   CamCalc.CrossChain_Cam[0..99].inflectionPointParameter := 0.5;
   CamCalc.CrossChain_Cam[0..99].modVeloTrapezoidParameter := 1.0;
   CamCalc.CrossChain_Cam[0..99].modSineMaxAccelCaStar := 0.0;
   CamCalc.CrossChain_Cam[0].camProfileType := 2;
   CamCalc.CrossChain_Cam[1..2].camProfileType := 1;
   CamCalc.CrossChain_Cam[3].camProfileType := 3;
   CamCalc.CrossChain_Cam[4..5].camProfileType := 1;
   CamCalc.CrossChain_Cam[6..99].camProfileType := 0;
   CamCalc.BeltChain_Cam[0..99].leadingValueStart := 0.0;
   CamCalc.BeltChain_Cam[0..99].leadingValueEnd := 0.0;
   CamCalc.BeltChain_Cam[0..99].followingValueStart := 0.0;
   CamCalc.BeltChain_Cam[0..99].followingValueEnd := 0.0;
   CamCalc.BeltChain_Cam[0..99].geoVeloStart := 0.0;
   CamCalc.BeltChain_Cam[0..99].geoVeloEnd := 0.0;
   CamCalc.BeltChain_Cam[0..99].geoAccelStart := 0.0;
   CamCalc.BeltChain_Cam[0..99].geoAccelEnd := 0.0;
   CamCalc.BeltChain_Cam[0..99].geoJerkStart := 0.0;
   CamCalc.BeltChain_Cam[0..99].geoJerkEnd := 0.0;
   CamCalc.BeltChain_Cam[0..99].inflectionPointParameter := 0.5;
   CamCalc.BeltChain_Cam[0..99].modVeloTrapezoidParameter := 1.0;
   CamCalc.BeltChain_Cam[0..99].modSineMaxAccelCaStar := 0.0;
   CamCalc.BeltChain_Cam[0..99].camProfileType := 0;
   CamCalc.ContChain_Cam[0..99].leadingValueStart := 0.0;
   CamCalc.ContChain_Cam[0].leadingValueEnd := 360.0;
   CamCalc.ContChain_Cam[1..99].leadingValueEnd := 0.0;
   CamCalc.ContChain_Cam[0..99].followingValueStart := 0.0;
   CamCalc.ContChain_Cam[0].followingValueEnd := 406.399993896484;
   CamCalc.ContChain_Cam[1..99].followingValueEnd := 0.0;
   CamCalc.ContChain_Cam[0..99].geoVeloStart := 0.0;
   CamCalc.ContChain_Cam[0..99].geoVeloEnd := 0.0;
   CamCalc.ContChain_Cam[0..99].geoAccelStart := 0.0;
   CamCalc.ContChain_Cam[0..99].geoAccelEnd := 0.0;
   CamCalc.ContChain_Cam[0..99].geoJerkStart := 0.0;
   CamCalc.ContChain_Cam[0..99].geoJerkEnd := 0.0;
   CamCalc.ContChain_Cam[0..99].inflectionPointParameter := 0.5;
   CamCalc.ContChain_Cam[0..99].modVeloTrapezoidParameter := 1.0;
   CamCalc.ContChain_Cam[0..99].modSineMaxAccelCaStar := 0.0;
   CamCalc.ContChain_Cam[0].camProfileType := 3;
   CamCalc.ContChain_Cam[1..99].camProfileType := 0;
   CamCalc.TransferChain_Cam[0..99].leadingValueStart := 0.0;
   CamCalc.TransferChain_Cam[0..99].leadingValueEnd := 0.0;
   CamCalc.TransferChain_Cam[0..99].followingValueStart := 0.0;
   CamCalc.TransferChain_Cam[0..99].followingValueEnd := 0.0;
   CamCalc.TransferChain_Cam[0..99].geoVeloStart := 0.0;
   CamCalc.TransferChain_Cam[0..99].geoVeloEnd := 0.0;
   CamCalc.TransferChain_Cam[0..99].geoAccelStart := 0.0;
   CamCalc.TransferChain_Cam[0..99].geoAccelEnd := 0.0;
   CamCalc.TransferChain_Cam[0..99].geoJerkStart := 0.0;
   CamCalc.TransferChain_Cam[0..99].geoJerkEnd := 0.0;
   CamCalc.TransferChain_Cam[0..99].inflectionPointParameter := 0.5;
   CamCalc.TransferChain_Cam[0..99].modVeloTrapezoidParameter := 1.0;
   CamCalc.TransferChain_Cam[0..99].modSineMaxAccelCaStar := 0.0;
   CamCalc.TransferChain_Cam[0..99].camProfileType := 0;
   CamCalc.ColumnAscChain_Cam[0..99].leadingValueStart := 0.0;
   CamCalc.ColumnAscChain_Cam[0..99].leadingValueEnd := 0.0;
   CamCalc.ColumnAscChain_Cam[0..99].followingValueStart := 0.0;
   CamCalc.ColumnAscChain_Cam[0..99].followingValueEnd := 0.0;
   CamCalc.ColumnAscChain_Cam[0..99].geoVeloStart := 0.0;
   CamCalc.ColumnAscChain_Cam[0..99].geoVeloEnd := 0.0;
   CamCalc.ColumnAscChain_Cam[0..99].geoAccelStart := 0.0;
   CamCalc.ColumnAscChain_Cam[0..99].geoAccelEnd := 0.0;
   CamCalc.ColumnAscChain_Cam[0..99].geoJerkStart := 0.0;
   CamCalc.ColumnAscChain_Cam[0..99].geoJerkEnd := 0.0;
   CamCalc.ColumnAscChain_Cam[0..99].inflectionPointParameter := 0.5;
   CamCalc.ColumnAscChain_Cam[0..99].modVeloTrapezoidParameter := 1.0;
   CamCalc.ColumnAscChain_Cam[0..99].modSineMaxAccelCaStar := 0.0;
   CamCalc.ColumnAscChain_Cam[0..99].camProfileType := 0;
   CamCalc.ColumnDescChain_Cam[0..99].leadingValueStart := 0.0;
   CamCalc.ColumnDescChain_Cam[0..99].leadingValueEnd := 0.0;
   CamCalc.ColumnDescChain_Cam[0..99].followingValueStart := 0.0;
   CamCalc.ColumnDescChain_Cam[0..99].followingValueEnd := 0.0;
   CamCalc.ColumnDescChain_Cam[0..99].geoVeloStart := 0.0;
   CamCalc.ColumnDescChain_Cam[0..99].geoVeloEnd := 0.0;
   CamCalc.ColumnDescChain_Cam[0..99].geoAccelStart := 0.0;
   CamCalc.ColumnDescChain_Cam[0..99].geoAccelEnd := 0.0;
   CamCalc.ColumnDescChain_Cam[0..99].geoJerkStart := 0.0;
   CamCalc.ColumnDescChain_Cam[0..99].geoJerkEnd := 0.0;
   CamCalc.ColumnDescChain_Cam[0..99].inflectionPointParameter := 0.5;
   CamCalc.ColumnDescChain_Cam[0..99].modVeloTrapezoidParameter := 1.0;
   CamCalc.ColumnDescChain_Cam[0..99].modSineMaxAccelCaStar := 0.0;
   CamCalc.ColumnDescChain_Cam[0..99].camProfileType := 0;
   CamCalc.CrossChain4_Cam[0].leadingValueStart := 0.0;
   CamCalc.CrossChain4_Cam[1].leadingValueStart := 193.679992675781;
   CamCalc.CrossChain4_Cam[2..3].leadingValueStart := 225.360000610352;
   CamCalc.CrossChain4_Cam[4].leadingValueStart := 328.320007324219;
   CamCalc.CrossChain4_Cam[5].leadingValueStart := 360.0;
   CamCalc.CrossChain4_Cam[6..99].leadingValueStart := 0.0;
   CamCalc.CrossChain4_Cam[0].leadingValueEnd := 162.0;
   CamCalc.CrossChain4_Cam[1..2].leadingValueEnd := 0.0;
   CamCalc.CrossChain4_Cam[3].leadingValueEnd := 296.640014648438;
   CamCalc.CrossChain4_Cam[4..99].leadingValueEnd := 0.0;
   CamCalc.CrossChain4_Cam[0].followingValueStart := 0.0;
   CamCalc.CrossChain4_Cam[1].followingValueStart := 31.8745098114014;
   CamCalc.CrossChain4_Cam[2..3].followingValueStart := 191.247055053711;
   CamCalc.CrossChain4_Cam[4].followingValueStart := 780.925476074219;
   CamCalc.CrossChain4_Cam[5].followingValueStart := 812.799987792969;
   CamCalc.CrossChain4_Cam[6..99].followingValueStart := 0.0;
   CamCalc.CrossChain4_Cam[0..2].followingValueEnd := 0.0;
   CamCalc.CrossChain4_Cam[3].followingValueEnd := 621.552917480469;
   CamCalc.CrossChain4_Cam[4..99].followingValueEnd := 0.0;
   CamCalc.CrossChain4_Cam[0..99].geoVeloStart := 0.0;
   CamCalc.CrossChain4_Cam[0..99].geoVeloEnd := 0.0;
   CamCalc.CrossChain4_Cam[0..99].geoAccelStart := 0.0;
   CamCalc.CrossChain4_Cam[0..99].geoAccelEnd := 0.0;
   CamCalc.CrossChain4_Cam[0..99].geoJerkStart := 0.0;
   CamCalc.CrossChain4_Cam[0..99].geoJerkEnd := 0.0;
   CamCalc.CrossChain4_Cam[0..99].inflectionPointParameter := 0.5;
   CamCalc.CrossChain4_Cam[0..99].modVeloTrapezoidParameter := 1.0;
   CamCalc.CrossChain4_Cam[0..99].modSineMaxAccelCaStar := 0.0;
   CamCalc.CrossChain4_Cam[0].camProfileType := 2;
   CamCalc.CrossChain4_Cam[1..2].camProfileType := 1;
   CamCalc.CrossChain4_Cam[3].camProfileType := 3;
   CamCalc.CrossChain4_Cam[4..5].camProfileType := 1;
   CamCalc.CrossChain4_Cam[6..99].camProfileType := 0;
   Chain1Long.AlmOk := TRUE;
   Chain1Long.StationWorked := TRUE;
   Chain1Long.CheckObstruction := TRUE;
   Chain1Long.OutChainObstruction := TRUE;
   Chain1Long.StrobeWork := FALSE;
   Chain1Long.StrobeShift := FALSE;
   Chain1Long.ManualMovement := FALSE;
   Chain1Long.OkToStop := TRUE;
   Chain1Long.PosOk := FALSE;
   Chain1Long.Ons_PosOk := FALSE;
   Chain1Long.EnaMove := TRUE;
   Chain1Long.StationEna := FALSE;
   Chain1Long.ModeLong := TRUE;
   Chain1Long.ModeCross := FALSE;
   Chain1Long.ModeCont := FALSE;
   Chain1Long.Cfg_Mould_ChainSteps := 1;
   Chain1Long.Cfg_Mould_EndPos := 38;
   Chain1Long.Shift_Lenght := 39;
   Chain1Long.PosMasterAdvanceStep := 0.0;
   Chain1Long.Input.EndChaMouPre := FALSE;
   Chain1Long.Input.PshHig := FALSE;
   Chain1Long.Input.PshLow := FALSE;
   Chain1Long.Output.PshHig := FALSE;
   Chain1Long.Output.PshLow := FALSE;
   Chain1Long.Man.EnaPbt := FALSE;
   Chain1Long.Man.RstCmd := TRUE;
   Chain1Long.Man.ScreenNumber := 300_010_301;
   Chain1Long.Man.WithinScreenRange := 0;
   Chain1Long.Drive.AlmOk := FALSE;
   Chain1Long.Drive.AlmEmerg := FALSE;
   Chain1Long.Drive.AlmNode := FALSE;
   Chain1Long.Drive.InitPosDrive := FALSE;
   Chain1Long.Drive.InitPosDrivePLS := FALSE;
   Chain1Long.Drive.GearingON := FALSE;
   Chain1Long.Drive.CamHook := FALSE;
   Chain1Long.Drive.CamStoppingPhase := FALSE;
   Chain1Long.Drive.RepositioningRequest := FALSE;
   Chain1Long.Drive.CamRequestResult := FALSE;
   Chain1Long.Drive.CamRequestError := FALSE;
   Chain1Long.Drive.CamRequestOk := TRUE;
   Chain1Long.Drive.CalibDisAxisReq := FALSE;
   Chain1Long.Drive.CalibReq := FALSE;
   Chain1Long.Drive.CalibProcess := FALSE;
   Chain1Long.Drive.HwOvertravelDisReq := FALSE;
   Chain1Long.Drive.HwOvertravelEnReq := FALSE;
   Chain1Long.Drive.AuxCamRequest := FALSE;
   Chain1Long.Drive.TorquePeakEna := TRUE;
   Chain1Long.Drive.Cmd_Repos := FALSE;
   Chain1Long.Drive.Ons_CamRequest := FALSE;
   Chain1Long.Drive.AuxCmdPosition := 0;
   Chain1Long.Drive.Unwind := 406.4;
   Chain1Long.Drive.MaxDev := 150.0;
   Chain1Long.Drive.ReposSpeed := 10.0;
   Chain1Long.Drive.CalcSlaveDifferenceABS := 0.0;
   Chain1Long.Drive.CalcModPosition := 0.0;
   Chain1Long.Drive.CalcSlaveDifference := 0.0;
   Chain1Long.Drive.CalcMinDeltaPos := 0.0;
   Chain1Long.Drive.CalcMaxDeltaPos := 0.0;
   Chain1Long.Drive.CalcHalfPosUnwind := 0.0;
   Chain1Long.Drive.Man.Cmd_PosJog := FALSE;
   Chain1Long.Drive.Man.Cmd_NegJog := FALSE;
   Chain1Long.Drive.Man.Cmd_Step := FALSE;
   Chain1Long.Drive.Man.Cmd_Forward := FALSE;
   Chain1Long.Drive.Man.Cmd_Backward := FALSE;
   Chain1Long.Drive.Man.Cmd_Up := FALSE;
   Chain1Long.Drive.Man.Cmd_Down := FALSE;
   Chain1Long.Drive.Man.Cmd_Intermediate := FALSE;
   Chain1Long.Drive.Man.Cmd_Open := FALSE;
   Chain1Long.Drive.Man.Cmd_Close := FALSE;
   Chain1Long.Drive.Man.Cmd_PreOpen := FALSE;
   Chain1Long.Drive.Man.Cmd_Maintenance := FALSE;
   Chain1Long.Drive.Man.Cmd_OperatorSide := FALSE;
   Chain1Long.Drive.Man.Cmd_NotOperatorSide := FALSE;
   Chain1Long.Drive.Man.Cmd_OnMould := FALSE;
   Chain1Long.Drive.Man.Cmd_OffMould := FALSE;
   Chain1Long.Drive.Man.Cmd_Pos0 := FALSE;
   Chain1Long.Drive.Man.Cmd_Pos1 := FALSE;
   Chain1Long.Drive.Man.Cmd_Pos2 := FALSE;
   Chain1Long.Drive.Man.Cmd_Pos3 := FALSE;
   Chain1Long.Drive.Man.Cmd_Pos4 := FALSE;
   Chain1Long.Drive.Man.Cmd_Pos5 := FALSE;
   Chain1Long.Drive.Man.Ons_Step := FALSE;
   Chain1Long.Drive.Man.PhaseJogCmd := FALSE;
   Chain1Long.Drive.Man.CmdStartStep := FALSE;
   Chain1Long.Drive.Man.CmdEndStep := FALSE;
   Chain1Long.Drive.Man.StepCond := FALSE;
   Chain1Long.Drive.Man.TON_DelayHomeCmd.PT := T#3S;
   Chain1Long.Drive.Man.TON_DelayHomeCmd.IN := FALSE;
   Chain1Long.Drive.Auto.Cmd_Step := FALSE;
   Chain1Long.Drive.Auto.Cmd_StartStep := FALSE;
   Chain1Long.Drive.Auto.Cmd_EndStep := FALSE;
   Chain1Long.Drive.Auto.Cmd_Forward := FALSE;
   Chain1Long.Drive.Auto.Cmd_Backward := FALSE;
   Chain1Long.Drive.Auto.Cmd_Up := FALSE;
   Chain1Long.Drive.Auto.Cmd_Down := FALSE;
   Chain1Long.Drive.Auto.Cmd_Intermediate := FALSE;
   Chain1Long.Drive.Auto.Cmd_Open := FALSE;
   Chain1Long.Drive.Auto.Cmd_Close := FALSE;
   Chain1Long.Drive.Auto.Cmd_PreOpen := FALSE;
   Chain1Long.Drive.Auto.Cmd_Maintenance := FALSE;
   Chain1Long.Drive.Auto.Cmd_OperatorSide := FALSE;
   Chain1Long.Drive.Auto.Cmd_NotOperatorSide := FALSE;
   Chain1Long.Drive.Auto.Cmd_OnMould := FALSE;
   Chain1Long.Drive.Auto.Cmd_OffMould := FALSE;
   Chain1Long.Drive.Auto.Cmd_Pos0 := FALSE;
   Chain1Long.Drive.Auto.Cmd_Pos1 := FALSE;
   Chain1Long.Drive.Auto.Cmd_Pos2 := FALSE;
   Chain1Long.Drive.Auto.Cmd_Pos3 := FALSE;
   Chain1Long.Drive.Auto.Cmd_Pos4 := FALSE;
   Chain1Long.Drive.Auto.Cmd_Pos5 := FALSE;
   Chain1Long.Drive.Auto.Cmd_Gear := FALSE;
   Chain1Long.Drive.ACT.CMD.Enable := FALSE;
   Chain1Long.Drive.ACT.CMD.Pos_Mode := FALSE;
   Chain1Long.Drive.ACT.CMD.MergeDisabled := FALSE;
   Chain1Long.Drive.ACT.CMD.SCurve := FALSE;
   Chain1Long.Drive.ACT.CMD.Cam_Mode := TRUE;
   Chain1Long.Drive.ACT.CMD.Cam_Request := FALSE;
   Chain1Long.Drive.ACT.CMD.Cam_PhaseStop := FALSE;
   Chain1Long.Drive.ACT.CMD.Gear_Mode := FALSE;
   Chain1Long.Drive.ACT.CMD.Repos_Req := FALSE;
   Chain1Long.Drive.ACT.CMD.Jog_Pos := FALSE;
   Chain1Long.Drive.ACT.CMD.Jog_Neg := FALSE;
   Chain1Long.Drive.ACT.CMD.Stop := FALSE;
   Chain1Long.Drive.ACT.CMD.Calibration_Req := FALSE;
   Chain1Long.Drive.ACT.CMD.Reset := FALSE;
   Chain1Long.Drive.ACT.CMD.RegInput1 := FALSE;
   Chain1Long.Drive.ACT.CMD.Brake_Release := FALSE;
   Chain1Long.Drive.ACT.CMD.HwPosOvertravel_Dis := FALSE;
   Chain1Long.Drive.ACT.CMD.HwNegOvertravel_Dis := FALSE;
   Chain1Long.Drive.ACT.CMD.HwOvertravel_MSG_En := FALSE;
   Chain1Long.Drive.ACT.CMD.OneShootMove := FALSE;
   Chain1Long.Drive.ACT.CMD.Move_Type := 3;
   Chain1Long.Drive.ACT.CMD.Target_Pos := 0.0;
   Chain1Long.Drive.ACT.CMD.Speed := 0.0;
   Chain1Long.Drive.ACT.CMD.Acceleration := 300.0;
   Chain1Long.Drive.ACT.CMD.Deceleration := 300.0;
   Chain1Long.Drive.ACT.CMD.Torque_Limit := 30.0;
   Chain1Long.Drive.ACT.CMD.Gear_Ratio := 0.0;
   Chain1Long.Drive.ACT.CMD.Mccp_Length := 2;
   Chain1Long.Drive.ACT.CMD.Mccp_StartSlope := 0.0;
   Chain1Long.Drive.ACT.CMD.Mccp_EndSlope := 0.0;
   Chain1Long.Drive.ACT.CMD.Mapc_Direction := 1;
   Chain1Long.Drive.ACT.CMD.Mapc_SlaveScaling := 1.0;
   Chain1Long.Drive.ACT.CMD.Mapc_MasterScaling := 1.0;
   Chain1Long.Drive.ACT.CMD.Mapc_MasterLockPosition := 0.0;
   Chain1Long.Drive.ACT.CMD.Mapc_CamLockPosition := 0.0;
   Chain1Long.Drive.ACT.CMD.Cam[0].leadingValueStart := 0.0;
   Chain1Long.Drive.ACT.CMD.Cam[1].leadingValueStart := 162.0;
   Chain1Long.Drive.ACT.CMD.Cam[2..39].leadingValueStart := 0.0;
   Chain1Long.Drive.ACT.CMD.Cam[0].leadingValueEnd := 162.0;
   Chain1Long.Drive.ACT.CMD.Cam[1].leadingValueEnd := 360.0;
   Chain1Long.Drive.ACT.CMD.Cam[2..39].leadingValueEnd := 0.0;
   Chain1Long.Drive.ACT.CMD.Cam[0].followingValueStart := 0.0;
   Chain1Long.Drive.ACT.CMD.Cam[1].followingValueStart := 406.399993896484;
   Chain1Long.Drive.ACT.CMD.Cam[2..39].followingValueStart := 0.0;
   Chain1Long.Drive.ACT.CMD.Cam[0..1].followingValueEnd := 406.399993896484;
   Chain1Long.Drive.ACT.CMD.Cam[2..39].followingValueEnd := 0.0;
   Chain1Long.Drive.ACT.CMD.Cam[0..39].geoVeloStart := 0.0;
   Chain1Long.Drive.ACT.CMD.Cam[0..39].geoVeloEnd := 0.0;
   Chain1Long.Drive.ACT.CMD.Cam[0..39].geoAccelStart := 0.0;
   Chain1Long.Drive.ACT.CMD.Cam[0..39].geoAccelEnd := 0.0;
   Chain1Long.Drive.ACT.CMD.Cam[0..39].geoJerkStart := 0.0;
   Chain1Long.Drive.ACT.CMD.Cam[0..39].geoJerkEnd := 0.0;
   Chain1Long.Drive.ACT.CMD.Cam[0..39].inflectionPointParameter := 0.5;
   Chain1Long.Drive.ACT.CMD.Cam[0..39].modVeloTrapezoidParameter := 1.0;
   Chain1Long.Drive.ACT.CMD.Cam[0..39].modSineMaxAccelCaStar := 0.0;
   Chain1Long.Drive.ACT.CMD.Cam[0].camProfileType := 5;
   Chain1Long.Drive.ACT.CMD.Cam[1].camProfileType := 2;
   Chain1Long.Drive.ACT.CMD.Cam[2..39].camProfileType := 0;
   Chain1Long.Drive.ACT.FBK.Ready := TRUE;
   Chain1Long.Drive.ACT.FBK.Calibrated := TRUE;
   Chain1Long.Drive.ACT.FBK.Fault := FALSE;
   Chain1Long.Drive.ACT.FBK.ModuleConnFault := FALSE;
   Chain1Long.Drive.ACT.FBK.In_Position := FALSE;
   Chain1Long.Drive.ACT.FBK.Standstill := TRUE;
   Chain1Long.Drive.ACT.FBK.Enabled := FALSE;
   Chain1Long.Drive.ACT.FBK.BusReadyStatus := FALSE;
   Chain1Long.Drive.ACT.FBK.BrakeReleased := FALSE;
   Chain1Long.Drive.ACT.FBK.HwPosOvertravelDisabled := FALSE;
   Chain1Long.Drive.ACT.FBK.HwNegOvertravelDisabled := FALSE;
   Chain1Long.Drive.ACT.FBK.SafeOffStatus := FALSE;
   Chain1Long.Drive.ACT.FBK.MaxTorqueLimit := FALSE;
   Chain1Long.Drive.ACT.FBK.PosMerge_IP := FALSE;
   Chain1Long.Drive.ACT.FBK.PosMerge_PC := FALSE;
   Chain1Long.Drive.ACT.FBK.Gearing_IP := FALSE;
   Chain1Long.Drive.ACT.FBK.Position := 279.321;
   Chain1Long.Drive.ACT.FBK.Speed := 0.0;
   Chain1Long.Drive.ACT.FBK.Torque := -0.006103516;
   Chain1Long.Drive.ACT.FBK.RegInput1Pos := 0.0;
   Chain1Long.Drive.ACT.FBK.SeqCamErrorCode := 0;
   Chain1Long.Drive.ACT.FBK.SeqCamTargetPosMAM := 0.0;
   Chain1Long.Drive.ACT.FBK.SeqCamStatus.EndSequence := FALSE;
   Chain1Long.Drive.ACT.FBK.SeqCamStatus.EndSuccess := FALSE;
   Chain1Long.Drive.ACT.FBK.SeqCamStatus.EndError := FALSE;
   Chain1Long.Drive.ACT.FBK.SeqCamStatus.CamHook := FALSE;
   Chain1Long.Drive.ACT.FBK.SeqCamStatus.BothMapc_IP := FALSE;
   Chain1Long.Drive.ACT.FBK.SeqCamStatus.SlaveFwd := FALSE;
   Chain1Long.Drive.ACT.FBK.SeqCamStatus.SlaveBwd := FALSE;
   Chain1Long.Drive.ACT.FBK.SeqCamStatus.SlaveUnwind := FALSE;
   Chain1Long.Drive.ACT.FBK.SeqCamStatus.WaitValidByOpe := FALSE;
   Chain1Long.Drive.ACT.FBK.SeqCamStatus.MapcA_IP := FALSE;
   Chain1Long.Drive.ACT.FBK.SeqCamStatus.MapcB_IP := FALSE;
   Chain1Long.Drive.ACT.FBK.SeqCamStatus.MapcC_IP := FALSE;
   Chain1Long.Drive.ACT.FBK.SeqCamStatus.CamOnce_PC := FALSE;
   Chain1Long.Drive.ACT.FBK.SeqCamStatus.MaxDevError := FALSE;
   Chain1Long.Drive.ACT.FBK.SeqCamStatus.PositionCamLockStatus := FALSE;
   Chain1Long.Drive.ACT.FBK.SeqCamStatus.WaitRestart := FALSE;
   Chain1Long.Drive.ACT.FBK.SeqCamStatus.Bit17 := FALSE;
   Chain1Long.Drive.ACT.FBK.SeqCamStatus.Bit18 := FALSE;
   Chain1Long.Drive.ACT.FBK.SeqCamStatus.Bit19 := FALSE;
   Chain1Long.Drive.ACT.FBK.SeqCamStatus.Bit20 := FALSE;
   Chain1Long.Drive.ACT.FBK.SeqCamStatus.Bit21 := FALSE;
   Chain1Long.Drive.ACT.FBK.SeqCamStatus.Bit22 := FALSE;
   Chain1Long.Drive.ACT.FBK.SeqCamStatus.Bit23 := FALSE;
   Chain1Long.Drive.ACT.FBK.SeqCamStatus.Bit24 := FALSE;
   Chain1Long.Drive.ACT.FBK.SeqCamStatus.Bit25 := FALSE;
   Chain1Long.Drive.ACT.FBK.SeqCamStatus.Bit26 := FALSE;
   Chain1Long.Drive.ACT.FBK.SeqCamStatus.Bit27 := FALSE;
   Chain1Long.Drive.ACT.FBK.SeqCamStatus.Bit28 := FALSE;
   Chain1Long.Drive.ACT.FBK.SeqCamStatus.Bit29 := FALSE;
   Chain1Long.Drive.ACT.FBK.SeqCamStatus.Bit30 := FALSE;
   Chain1Long.Drive.ACT.FBK.SeqCamStatus.Bit31 := FALSE;
   Chain1Long.Drive.ACT.FBK.SeqCamStatus.Bit32 := FALSE;
   Chain1Long.Drive.PLS.FinePosOk.LowLimit := 405.4;
   Chain1Long.Drive.PLS.FinePosOk.HighLimit := 1.0;
   Chain1Long.Drive.PLS.FinePosOk.Ok := FALSE;
   Chain1Long.Drive.PLS.KeepPosOk.LowLimit := 404.4;
   Chain1Long.Drive.PLS.KeepPosOk.HighLimit := 2.0;
   Chain1Long.Drive.PLS.KeepPosOk.Ok := FALSE;
   Chain1Long.Drive.PLS.Up.LowLimit := 0.0;
   Chain1Long.Drive.PLS.Up.HighLimit := 0.0;
   Chain1Long.Drive.PLS.Up.Ok := FALSE;
   Chain1Long.Drive.PLS.Intermediate.LowLimit := 0.0;
   Chain1Long.Drive.PLS.Intermediate.HighLimit := 0.0;
   Chain1Long.Drive.PLS.Intermediate.Ok := FALSE;
   Chain1Long.Drive.PLS.Down.LowLimit := 0.0;
   Chain1Long.Drive.PLS.Down.HighLimit := 0.0;
   Chain1Long.Drive.PLS.Down.Ok := FALSE;
   Chain1Long.Drive.PLS.Forward.LowLimit := 0.0;
   Chain1Long.Drive.PLS.Forward.HighLimit := 0.0;
   Chain1Long.Drive.PLS.Forward.Ok := FALSE;
   Chain1Long.Drive.PLS.Backward.LowLimit := 0.0;
   Chain1Long.Drive.PLS.Backward.HighLimit := 0.0;
   Chain1Long.Drive.PLS.Backward.Ok := FALSE;
   Chain1Long.Drive.PLS.Open.LowLimit := 0.0;
   Chain1Long.Drive.PLS.Open.HighLimit := 0.0;
   Chain1Long.Drive.PLS.Open.Ok := FALSE;
   Chain1Long.Drive.PLS.Close.LowLimit := 0.0;
   Chain1Long.Drive.PLS.Close.HighLimit := 0.0;
   Chain1Long.Drive.PLS.Close.Ok := FALSE;
   Chain1Long.Drive.PLS.PreOpen.LowLimit := 0.0;
   Chain1Long.Drive.PLS.PreOpen.HighLimit := 0.0;
   Chain1Long.Drive.PLS.PreOpen.Ok := FALSE;
   Chain1Long.Drive.PLS.Maintenance.LowLimit := 0.0;
   Chain1Long.Drive.PLS.Maintenance.HighLimit := 0.0;
   Chain1Long.Drive.PLS.Maintenance.Ok := FALSE;
   Chain1Long.Drive.PLS.OperatorSide.LowLimit := 0.0;
   Chain1Long.Drive.PLS.OperatorSide.HighLimit := 0.0;
   Chain1Long.Drive.PLS.OperatorSide.Ok := FALSE;
   Chain1Long.Drive.PLS.NotOperatorSide.LowLimit := 0.0;
   Chain1Long.Drive.PLS.NotOperatorSide.HighLimit := 0.0;
   Chain1Long.Drive.PLS.NotOperatorSide.Ok := FALSE;
   Chain1Long.Drive.PLS.OnMould.LowLimit := 0.0;
   Chain1Long.Drive.PLS.OnMould.HighLimit := 0.0;
   Chain1Long.Drive.PLS.OnMould.Ok := FALSE;
   Chain1Long.Drive.PLS.OffMould.LowLimit := 0.0;
   Chain1Long.Drive.PLS.OffMould.HighLimit := 0.0;
   Chain1Long.Drive.PLS.OffMould.Ok := FALSE;
   Chain1Long.Drive.PLS.Pos0.LowLimit := 0.0;
   Chain1Long.Drive.PLS.Pos0.HighLimit := 0.0;
   Chain1Long.Drive.PLS.Pos0.Ok := FALSE;
   Chain1Long.Drive.PLS.Pos1.LowLimit := 0.0;
   Chain1Long.Drive.PLS.Pos1.HighLimit := 0.0;
   Chain1Long.Drive.PLS.Pos1.Ok := FALSE;
   Chain1Long.Drive.PLS.Pos2.LowLimit := 0.0;
   Chain1Long.Drive.PLS.Pos2.HighLimit := 0.0;
   Chain1Long.Drive.PLS.Pos2.Ok := FALSE;
   Chain1Long.Drive.PLS.Pos3.LowLimit := 0.0;
   Chain1Long.Drive.PLS.Pos3.HighLimit := 0.0;
   Chain1Long.Drive.PLS.Pos3.Ok := FALSE;
   Chain1Long.Drive.PLS.Pos4.LowLimit := 0.0;
   Chain1Long.Drive.PLS.Pos4.HighLimit := 0.0;
   Chain1Long.Drive.PLS.Pos4.Ok := FALSE;
   Chain1Long.Drive.PLS.Pos5.LowLimit := 0.0;
   Chain1Long.Drive.PLS.Pos5.HighLimit := 0.0;
   Chain1Long.Drive.PLS.Pos5.Ok := FALSE;
   Chain1Long.Drive.TON_EnableDrive.PT := T#500MS;
   Chain1Long.Drive.TON_EnableDrive.IN := FALSE;
   Chain1Long.Drive.TON_HwOvertravel_Dis.PT := T#0MS;
   Chain1Long.Drive.TON_HwOvertravel_Dis.IN := FALSE;
   Chain1Long.Drive.TON_HwOvertravel_En.PT := T#0MS;
   Chain1Long.Drive.TON_HwOvertravel_En.IN := FALSE;
   Chain1Long.Drive.TON_TimeoutMovement.PT := T#0MS;
   Chain1Long.Drive.TON_TimeoutMovement.IN := FALSE;
   Chain2Long.AlmOk := TRUE;
   Chain2Long.StationWorked := TRUE;
   Chain2Long.CheckObstruction := TRUE;
   Chain2Long.OutChainObstruction := TRUE;
   Chain2Long.StrobeWork := FALSE;
   Chain2Long.StrobeShift := FALSE;
   Chain2Long.ManualMovement := FALSE;
   Chain2Long.OkToStop := TRUE;
   Chain2Long.PosOk := FALSE;
   Chain2Long.Ons_PosOk := FALSE;
   Chain2Long.EnaMove := TRUE;
   Chain2Long.StationEna := FALSE;
   Chain2Long.ModeLong := TRUE;
   Chain2Long.ModeCross := FALSE;
   Chain2Long.ModeCont := FALSE;
   Chain2Long.Cfg_Mould_ChainSteps := 1;
   Chain2Long.Cfg_Mould_EndPos := 33;
   Chain2Long.Shift_Lenght := 34;
   Chain2Long.PosMasterAdvanceStep := 0.0;
   Chain2Long.Input.EndChaMouPre := FALSE;
   Chain2Long.Input.PshHig := FALSE;
   Chain2Long.Input.PshLow := FALSE;
   Chain2Long.Output.PshHig := FALSE;
   Chain2Long.Output.PshLow := FALSE;
   Chain2Long.Man.EnaPbt := FALSE;
   Chain2Long.Man.RstCmd := TRUE;
   Chain2Long.Man.ScreenNumber := 300_020_301;
   Chain2Long.Man.WithinScreenRange := 0;
   Chain2Long.Drive.AlmOk := FALSE;
   Chain2Long.Drive.AlmEmerg := FALSE;
   Chain2Long.Drive.AlmNode := FALSE;
   Chain2Long.Drive.InitPosDrive := FALSE;
   Chain2Long.Drive.InitPosDrivePLS := FALSE;
   Chain2Long.Drive.GearingON := FALSE;
   Chain2Long.Drive.CamHook := FALSE;
   Chain2Long.Drive.CamStoppingPhase := FALSE;
   Chain2Long.Drive.RepositioningRequest := FALSE;
   Chain2Long.Drive.CamRequestResult := FALSE;
   Chain2Long.Drive.CamRequestError := FALSE;
   Chain2Long.Drive.CamRequestOk := TRUE;
   Chain2Long.Drive.CalibDisAxisReq := FALSE;
   Chain2Long.Drive.CalibReq := FALSE;
   Chain2Long.Drive.CalibProcess := FALSE;
   Chain2Long.Drive.HwOvertravelDisReq := FALSE;
   Chain2Long.Drive.HwOvertravelEnReq := FALSE;
   Chain2Long.Drive.AuxCamRequest := FALSE;
   Chain2Long.Drive.TorquePeakEna := TRUE;
   Chain2Long.Drive.Cmd_Repos := FALSE;
   Chain2Long.Drive.Ons_CamRequest := FALSE;
   Chain2Long.Drive.AuxCmdPosition := 0;
   Chain2Long.Drive.Unwind := 406.4;
   Chain2Long.Drive.MaxDev := 150.0;
   Chain2Long.Drive.ReposSpeed := 10.0;
   Chain2Long.Drive.CalcSlaveDifferenceABS := 0.0;
   Chain2Long.Drive.CalcModPosition := 0.0;
   Chain2Long.Drive.CalcSlaveDifference := 0.0;
   Chain2Long.Drive.CalcMinDeltaPos := 0.0;
   Chain2Long.Drive.CalcMaxDeltaPos := 0.0;
   Chain2Long.Drive.CalcHalfPosUnwind := 0.0;
   Chain2Long.Drive.Man.Cmd_PosJog := FALSE;
   Chain2Long.Drive.Man.Cmd_NegJog := FALSE;
   Chain2Long.Drive.Man.Cmd_Step := FALSE;
   Chain2Long.Drive.Man.Cmd_Forward := FALSE;
   Chain2Long.Drive.Man.Cmd_Backward := FALSE;
   Chain2Long.Drive.Man.Cmd_Up := FALSE;
   Chain2Long.Drive.Man.Cmd_Down := FALSE;
   Chain2Long.Drive.Man.Cmd_Intermediate := FALSE;
   Chain2Long.Drive.Man.Cmd_Open := FALSE;
   Chain2Long.Drive.Man.Cmd_Close := FALSE;
   Chain2Long.Drive.Man.Cmd_PreOpen := FALSE;
   Chain2Long.Drive.Man.Cmd_Maintenance := FALSE;
   Chain2Long.Drive.Man.Cmd_OperatorSide := FALSE;
   Chain2Long.Drive.Man.Cmd_NotOperatorSide := FALSE;
   Chain2Long.Drive.Man.Cmd_OnMould := FALSE;
   Chain2Long.Drive.Man.Cmd_OffMould := FALSE;
   Chain2Long.Drive.Man.Cmd_Pos0 := FALSE;
   Chain2Long.Drive.Man.Cmd_Pos1 := FALSE;
   Chain2Long.Drive.Man.Cmd_Pos2 := FALSE;
   Chain2Long.Drive.Man.Cmd_Pos3 := FALSE;
   Chain2Long.Drive.Man.Cmd_Pos4 := FALSE;
   Chain2Long.Drive.Man.Cmd_Pos5 := FALSE;
   Chain2Long.Drive.Man.Ons_Step := FALSE;
   Chain2Long.Drive.Man.PhaseJogCmd := FALSE;
   Chain2Long.Drive.Man.CmdStartStep := FALSE;
   Chain2Long.Drive.Man.CmdEndStep := FALSE;
   Chain2Long.Drive.Man.StepCond := FALSE;
   Chain2Long.Drive.Man.TON_DelayHomeCmd.PT := T#3S;
   Chain2Long.Drive.Man.TON_DelayHomeCmd.IN := FALSE;
   Chain2Long.Drive.Auto.Cmd_Step := FALSE;
   Chain2Long.Drive.Auto.Cmd_StartStep := FALSE;
   Chain2Long.Drive.Auto.Cmd_EndStep := FALSE;
   Chain2Long.Drive.Auto.Cmd_Forward := FALSE;
   Chain2Long.Drive.Auto.Cmd_Backward := FALSE;
   Chain2Long.Drive.Auto.Cmd_Up := FALSE;
   Chain2Long.Drive.Auto.Cmd_Down := FALSE;
   Chain2Long.Drive.Auto.Cmd_Intermediate := FALSE;
   Chain2Long.Drive.Auto.Cmd_Open := FALSE;
   Chain2Long.Drive.Auto.Cmd_Close := FALSE;
   Chain2Long.Drive.Auto.Cmd_PreOpen := FALSE;
   Chain2Long.Drive.Auto.Cmd_Maintenance := FALSE;
   Chain2Long.Drive.Auto.Cmd_OperatorSide := FALSE;
   Chain2Long.Drive.Auto.Cmd_NotOperatorSide := FALSE;
   Chain2Long.Drive.Auto.Cmd_OnMould := FALSE;
   Chain2Long.Drive.Auto.Cmd_OffMould := FALSE;
   Chain2Long.Drive.Auto.Cmd_Pos0 := FALSE;
   Chain2Long.Drive.Auto.Cmd_Pos1 := FALSE;
   Chain2Long.Drive.Auto.Cmd_Pos2 := FALSE;
   Chain2Long.Drive.Auto.Cmd_Pos3 := FALSE;
   Chain2Long.Drive.Auto.Cmd_Pos4 := FALSE;
   Chain2Long.Drive.Auto.Cmd_Pos5 := FALSE;
   Chain2Long.Drive.Auto.Cmd_Gear := FALSE;
   Chain2Long.Drive.ACT.CMD.Enable := FALSE;
   Chain2Long.Drive.ACT.CMD.Pos_Mode := FALSE;
   Chain2Long.Drive.ACT.CMD.MergeDisabled := FALSE;
   Chain2Long.Drive.ACT.CMD.SCurve := FALSE;
   Chain2Long.Drive.ACT.CMD.Cam_Mode := TRUE;
   Chain2Long.Drive.ACT.CMD.Cam_Request := FALSE;
   Chain2Long.Drive.ACT.CMD.Cam_PhaseStop := FALSE;
   Chain2Long.Drive.ACT.CMD.Gear_Mode := FALSE;
   Chain2Long.Drive.ACT.CMD.Repos_Req := FALSE;
   Chain2Long.Drive.ACT.CMD.Jog_Pos := FALSE;
   Chain2Long.Drive.ACT.CMD.Jog_Neg := FALSE;
   Chain2Long.Drive.ACT.CMD.Stop := FALSE;
   Chain2Long.Drive.ACT.CMD.Calibration_Req := FALSE;
   Chain2Long.Drive.ACT.CMD.Reset := FALSE;
   Chain2Long.Drive.ACT.CMD.RegInput1 := FALSE;
   Chain2Long.Drive.ACT.CMD.Brake_Release := FALSE;
   Chain2Long.Drive.ACT.CMD.HwPosOvertravel_Dis := FALSE;
   Chain2Long.Drive.ACT.CMD.HwNegOvertravel_Dis := FALSE;
   Chain2Long.Drive.ACT.CMD.HwOvertravel_MSG_En := FALSE;
   Chain2Long.Drive.ACT.CMD.OneShootMove := FALSE;
   Chain2Long.Drive.ACT.CMD.Move_Type := 3;
   Chain2Long.Drive.ACT.CMD.Target_Pos := 0.0;
   Chain2Long.Drive.ACT.CMD.Speed := 0.0;
   Chain2Long.Drive.ACT.CMD.Acceleration := 300.0;
   Chain2Long.Drive.ACT.CMD.Deceleration := 300.0;
   Chain2Long.Drive.ACT.CMD.Torque_Limit := 30.0;
   Chain2Long.Drive.ACT.CMD.Gear_Ratio := 0.0;
   Chain2Long.Drive.ACT.CMD.Mccp_Length := 2;
   Chain2Long.Drive.ACT.CMD.Mccp_StartSlope := 0.0;
   Chain2Long.Drive.ACT.CMD.Mccp_EndSlope := 0.0;
   Chain2Long.Drive.ACT.CMD.Mapc_Direction := 1;
   Chain2Long.Drive.ACT.CMD.Mapc_SlaveScaling := 1.0;
   Chain2Long.Drive.ACT.CMD.Mapc_MasterScaling := 1.0;
   Chain2Long.Drive.ACT.CMD.Mapc_MasterLockPosition := 0.0;
   Chain2Long.Drive.ACT.CMD.Mapc_CamLockPosition := 0.0;
   Chain2Long.Drive.ACT.CMD.Cam[0].leadingValueStart := 0.0;
   Chain2Long.Drive.ACT.CMD.Cam[1].leadingValueStart := 162.0;
   Chain2Long.Drive.ACT.CMD.Cam[2..39].leadingValueStart := 0.0;
   Chain2Long.Drive.ACT.CMD.Cam[0].leadingValueEnd := 162.0;
   Chain2Long.Drive.ACT.CMD.Cam[1].leadingValueEnd := 360.0;
   Chain2Long.Drive.ACT.CMD.Cam[2..39].leadingValueEnd := 0.0;
   Chain2Long.Drive.ACT.CMD.Cam[0].followingValueStart := 0.0;
   Chain2Long.Drive.ACT.CMD.Cam[1].followingValueStart := 406.399993896484;
   Chain2Long.Drive.ACT.CMD.Cam[2..39].followingValueStart := 0.0;
   Chain2Long.Drive.ACT.CMD.Cam[0..1].followingValueEnd := 406.399993896484;
   Chain2Long.Drive.ACT.CMD.Cam[2..39].followingValueEnd := 0.0;
   Chain2Long.Drive.ACT.CMD.Cam[0..39].geoVeloStart := 0.0;
   Chain2Long.Drive.ACT.CMD.Cam[0..39].geoVeloEnd := 0.0;
   Chain2Long.Drive.ACT.CMD.Cam[0..39].geoAccelStart := 0.0;
   Chain2Long.Drive.ACT.CMD.Cam[0..39].geoAccelEnd := 0.0;
   Chain2Long.Drive.ACT.CMD.Cam[0..39].geoJerkStart := 0.0;
   Chain2Long.Drive.ACT.CMD.Cam[0..39].geoJerkEnd := 0.0;
   Chain2Long.Drive.ACT.CMD.Cam[0..39].inflectionPointParameter := 0.5;
   Chain2Long.Drive.ACT.CMD.Cam[0..39].modVeloTrapezoidParameter := 1.0;
   Chain2Long.Drive.ACT.CMD.Cam[0..39].modSineMaxAccelCaStar := 0.0;
   Chain2Long.Drive.ACT.CMD.Cam[0].camProfileType := 5;
   Chain2Long.Drive.ACT.CMD.Cam[1].camProfileType := 2;
   Chain2Long.Drive.ACT.CMD.Cam[2..39].camProfileType := 0;
   Chain2Long.Drive.ACT.FBK.Ready := TRUE;
   Chain2Long.Drive.ACT.FBK.Calibrated := TRUE;
   Chain2Long.Drive.ACT.FBK.Fault := FALSE;
   Chain2Long.Drive.ACT.FBK.ModuleConnFault := FALSE;
   Chain2Long.Drive.ACT.FBK.In_Position := FALSE;
   Chain2Long.Drive.ACT.FBK.Standstill := TRUE;
   Chain2Long.Drive.ACT.FBK.Enabled := FALSE;
   Chain2Long.Drive.ACT.FBK.BusReadyStatus := FALSE;
   Chain2Long.Drive.ACT.FBK.BrakeReleased := FALSE;
   Chain2Long.Drive.ACT.FBK.HwPosOvertravelDisabled := FALSE;
   Chain2Long.Drive.ACT.FBK.HwNegOvertravelDisabled := FALSE;
   Chain2Long.Drive.ACT.FBK.SafeOffStatus := FALSE;
   Chain2Long.Drive.ACT.FBK.MaxTorqueLimit := FALSE;
   Chain2Long.Drive.ACT.FBK.PosMerge_IP := FALSE;
   Chain2Long.Drive.ACT.FBK.PosMerge_PC := FALSE;
   Chain2Long.Drive.ACT.FBK.Gearing_IP := FALSE;
   Chain2Long.Drive.ACT.FBK.Position := 279.433;
   Chain2Long.Drive.ACT.FBK.Speed := 0.0;
   Chain2Long.Drive.ACT.FBK.Torque := 0.0;
   Chain2Long.Drive.ACT.FBK.RegInput1Pos := 0.0;
   Chain2Long.Drive.ACT.FBK.SeqCamErrorCode := 0;
   Chain2Long.Drive.ACT.FBK.SeqCamTargetPosMAM := 0.0;
   Chain2Long.Drive.ACT.FBK.SeqCamStatus.EndSequence := FALSE;
   Chain2Long.Drive.ACT.FBK.SeqCamStatus.EndSuccess := FALSE;
   Chain2Long.Drive.ACT.FBK.SeqCamStatus.EndError := FALSE;
   Chain2Long.Drive.ACT.FBK.SeqCamStatus.CamHook := FALSE;
   Chain2Long.Drive.ACT.FBK.SeqCamStatus.BothMapc_IP := FALSE;
   Chain2Long.Drive.ACT.FBK.SeqCamStatus.SlaveFwd := FALSE;
   Chain2Long.Drive.ACT.FBK.SeqCamStatus.SlaveBwd := FALSE;
   Chain2Long.Drive.ACT.FBK.SeqCamStatus.SlaveUnwind := FALSE;
   Chain2Long.Drive.ACT.FBK.SeqCamStatus.WaitValidByOpe := FALSE;
   Chain2Long.Drive.ACT.FBK.SeqCamStatus.MapcA_IP := FALSE;
   Chain2Long.Drive.ACT.FBK.SeqCamStatus.MapcB_IP := FALSE;
   Chain2Long.Drive.ACT.FBK.SeqCamStatus.MapcC_IP := FALSE;
   Chain2Long.Drive.ACT.FBK.SeqCamStatus.CamOnce_PC := FALSE;
   Chain2Long.Drive.ACT.FBK.SeqCamStatus.MaxDevError := FALSE;
   Chain2Long.Drive.ACT.FBK.SeqCamStatus.PositionCamLockStatus := FALSE;
   Chain2Long.Drive.ACT.FBK.SeqCamStatus.WaitRestart := FALSE;
   Chain2Long.Drive.ACT.FBK.SeqCamStatus.Bit17 := FALSE;
   Chain2Long.Drive.ACT.FBK.SeqCamStatus.Bit18 := FALSE;
   Chain2Long.Drive.ACT.FBK.SeqCamStatus.Bit19 := FALSE;
   Chain2Long.Drive.ACT.FBK.SeqCamStatus.Bit20 := FALSE;
   Chain2Long.Drive.ACT.FBK.SeqCamStatus.Bit21 := FALSE;
   Chain2Long.Drive.ACT.FBK.SeqCamStatus.Bit22 := FALSE;
   Chain2Long.Drive.ACT.FBK.SeqCamStatus.Bit23 := FALSE;
   Chain2Long.Drive.ACT.FBK.SeqCamStatus.Bit24 := FALSE;
   Chain2Long.Drive.ACT.FBK.SeqCamStatus.Bit25 := FALSE;
   Chain2Long.Drive.ACT.FBK.SeqCamStatus.Bit26 := FALSE;
   Chain2Long.Drive.ACT.FBK.SeqCamStatus.Bit27 := FALSE;
   Chain2Long.Drive.ACT.FBK.SeqCamStatus.Bit28 := FALSE;
   Chain2Long.Drive.ACT.FBK.SeqCamStatus.Bit29 := FALSE;
   Chain2Long.Drive.ACT.FBK.SeqCamStatus.Bit30 := FALSE;
   Chain2Long.Drive.ACT.FBK.SeqCamStatus.Bit31 := FALSE;
   Chain2Long.Drive.ACT.FBK.SeqCamStatus.Bit32 := FALSE;
   Chain2Long.Drive.PLS.FinePosOk.LowLimit := 405.4;
   Chain2Long.Drive.PLS.FinePosOk.HighLimit := 1.0;
   Chain2Long.Drive.PLS.FinePosOk.Ok := FALSE;
   Chain2Long.Drive.PLS.KeepPosOk.LowLimit := 404.4;
   Chain2Long.Drive.PLS.KeepPosOk.HighLimit := 2.0;
   Chain2Long.Drive.PLS.KeepPosOk.Ok := FALSE;
   Chain2Long.Drive.PLS.Up.LowLimit := 0.0;
   Chain2Long.Drive.PLS.Up.HighLimit := 0.0;
   Chain2Long.Drive.PLS.Up.Ok := FALSE;
   Chain2Long.Drive.PLS.Intermediate.LowLimit := 0.0;
   Chain2Long.Drive.PLS.Intermediate.HighLimit := 0.0;
   Chain2Long.Drive.PLS.Intermediate.Ok := FALSE;
   Chain2Long.Drive.PLS.Down.LowLimit := 0.0;
   Chain2Long.Drive.PLS.Down.HighLimit := 0.0;
   Chain2Long.Drive.PLS.Down.Ok := FALSE;
   Chain2Long.Drive.PLS.Forward.LowLimit := 0.0;
   Chain2Long.Drive.PLS.Forward.HighLimit := 0.0;
   Chain2Long.Drive.PLS.Forward.Ok := FALSE;
   Chain2Long.Drive.PLS.Backward.LowLimit := 0.0;
   Chain2Long.Drive.PLS.Backward.HighLimit := 0.0;
   Chain2Long.Drive.PLS.Backward.Ok := FALSE;
   Chain2Long.Drive.PLS.Open.LowLimit := 0.0;
   Chain2Long.Drive.PLS.Open.HighLimit := 0.0;
   Chain2Long.Drive.PLS.Open.Ok := FALSE;
   Chain2Long.Drive.PLS.Close.LowLimit := 0.0;
   Chain2Long.Drive.PLS.Close.HighLimit := 0.0;
   Chain2Long.Drive.PLS.Close.Ok := FALSE;
   Chain2Long.Drive.PLS.PreOpen.LowLimit := 0.0;
   Chain2Long.Drive.PLS.PreOpen.HighLimit := 0.0;
   Chain2Long.Drive.PLS.PreOpen.Ok := FALSE;
   Chain2Long.Drive.PLS.Maintenance.LowLimit := 0.0;
   Chain2Long.Drive.PLS.Maintenance.HighLimit := 0.0;
   Chain2Long.Drive.PLS.Maintenance.Ok := FALSE;
   Chain2Long.Drive.PLS.OperatorSide.LowLimit := 0.0;
   Chain2Long.Drive.PLS.OperatorSide.HighLimit := 0.0;
   Chain2Long.Drive.PLS.OperatorSide.Ok := FALSE;
   Chain2Long.Drive.PLS.NotOperatorSide.LowLimit := 0.0;
   Chain2Long.Drive.PLS.NotOperatorSide.HighLimit := 0.0;
   Chain2Long.Drive.PLS.NotOperatorSide.Ok := FALSE;
   Chain2Long.Drive.PLS.OnMould.LowLimit := 0.0;
   Chain2Long.Drive.PLS.OnMould.HighLimit := 0.0;
   Chain2Long.Drive.PLS.OnMould.Ok := FALSE;
   Chain2Long.Drive.PLS.OffMould.LowLimit := 0.0;
   Chain2Long.Drive.PLS.OffMould.HighLimit := 0.0;
   Chain2Long.Drive.PLS.OffMould.Ok := FALSE;
   Chain2Long.Drive.PLS.Pos0.LowLimit := 0.0;
   Chain2Long.Drive.PLS.Pos0.HighLimit := 0.0;
   Chain2Long.Drive.PLS.Pos0.Ok := FALSE;
   Chain2Long.Drive.PLS.Pos1.LowLimit := 0.0;
   Chain2Long.Drive.PLS.Pos1.HighLimit := 0.0;
   Chain2Long.Drive.PLS.Pos1.Ok := FALSE;
   Chain2Long.Drive.PLS.Pos2.LowLimit := 0.0;
   Chain2Long.Drive.PLS.Pos2.HighLimit := 0.0;
   Chain2Long.Drive.PLS.Pos2.Ok := FALSE;
   Chain2Long.Drive.PLS.Pos3.LowLimit := 0.0;
   Chain2Long.Drive.PLS.Pos3.HighLimit := 0.0;
   Chain2Long.Drive.PLS.Pos3.Ok := FALSE;
   Chain2Long.Drive.PLS.Pos4.LowLimit := 0.0;
   Chain2Long.Drive.PLS.Pos4.HighLimit := 0.0;
   Chain2Long.Drive.PLS.Pos4.Ok := FALSE;
   Chain2Long.Drive.PLS.Pos5.LowLimit := 0.0;
   Chain2Long.Drive.PLS.Pos5.HighLimit := 0.0;
   Chain2Long.Drive.PLS.Pos5.Ok := FALSE;
   Chain2Long.Drive.TON_EnableDrive.PT := T#500MS;
   Chain2Long.Drive.TON_EnableDrive.IN := FALSE;
   Chain2Long.Drive.TON_HwOvertravel_Dis.PT := T#0MS;
   Chain2Long.Drive.TON_HwOvertravel_Dis.IN := FALSE;
   Chain2Long.Drive.TON_HwOvertravel_En.PT := T#0MS;
   Chain2Long.Drive.TON_HwOvertravel_En.IN := FALSE;
   Chain2Long.Drive.TON_TimeoutMovement.PT := T#0MS;
   Chain2Long.Drive.TON_TimeoutMovement.IN := FALSE;
   Chain3Long.AlmOk := TRUE;
   Chain3Long.StationWorked := TRUE;
   Chain3Long.CheckObstruction := TRUE;
   Chain3Long.OutChainObstruction := TRUE;
   Chain3Long.StrobeWork := FALSE;
   Chain3Long.StrobeShift := FALSE;
   Chain3Long.ManualMovement := FALSE;
   Chain3Long.OkToStop := TRUE;
   Chain3Long.PosOk := FALSE;
   Chain3Long.Ons_PosOk := FALSE;
   Chain3Long.EnaMove := TRUE;
   Chain3Long.StationEna := FALSE;
   Chain3Long.ModeLong := TRUE;
   Chain3Long.ModeCross := FALSE;
   Chain3Long.ModeCont := FALSE;
   Chain3Long.Cfg_Mould_ChainSteps := 1;
   Chain3Long.Cfg_Mould_EndPos := 50;
   Chain3Long.Shift_Lenght := 51;
   Chain3Long.PosMasterAdvanceStep := 0.0;
   Chain3Long.Input.EndChaMouPre := FALSE;
   Chain3Long.Input.PshHig := FALSE;
   Chain3Long.Input.PshLow := FALSE;
   Chain3Long.Output.PshHig := FALSE;
   Chain3Long.Output.PshLow := FALSE;
   Chain3Long.Man.EnaPbt := FALSE;
   Chain3Long.Man.RstCmd := TRUE;
   Chain3Long.Man.ScreenNumber := 300_030_301;
   Chain3Long.Man.WithinScreenRange := 0;
   Chain3Long.Drive.AlmOk := FALSE;
   Chain3Long.Drive.AlmEmerg := FALSE;
   Chain3Long.Drive.AlmNode := FALSE;
   Chain3Long.Drive.InitPosDrive := FALSE;
   Chain3Long.Drive.InitPosDrivePLS := FALSE;
   Chain3Long.Drive.GearingON := FALSE;
   Chain3Long.Drive.CamHook := FALSE;
   Chain3Long.Drive.CamStoppingPhase := FALSE;
   Chain3Long.Drive.RepositioningRequest := FALSE;
   Chain3Long.Drive.CamRequestResult := FALSE;
   Chain3Long.Drive.CamRequestError := FALSE;
   Chain3Long.Drive.CamRequestOk := TRUE;
   Chain3Long.Drive.CalibDisAxisReq := FALSE;
   Chain3Long.Drive.CalibReq := FALSE;
   Chain3Long.Drive.CalibProcess := FALSE;
   Chain3Long.Drive.HwOvertravelDisReq := FALSE;
   Chain3Long.Drive.HwOvertravelEnReq := FALSE;
   Chain3Long.Drive.AuxCamRequest := FALSE;
   Chain3Long.Drive.TorquePeakEna := TRUE;
   Chain3Long.Drive.Cmd_Repos := FALSE;
   Chain3Long.Drive.Ons_CamRequest := FALSE;
   Chain3Long.Drive.AuxCmdPosition := 0;
   Chain3Long.Drive.Unwind := 406.4;
   Chain3Long.Drive.MaxDev := 150.0;
   Chain3Long.Drive.ReposSpeed := 10.0;
   Chain3Long.Drive.CalcSlaveDifferenceABS := 0.0;
   Chain3Long.Drive.CalcModPosition := 0.0;
   Chain3Long.Drive.CalcSlaveDifference := 0.0;
   Chain3Long.Drive.CalcMinDeltaPos := 0.0;
   Chain3Long.Drive.CalcMaxDeltaPos := 0.0;
   Chain3Long.Drive.CalcHalfPosUnwind := 0.0;
   Chain3Long.Drive.Man.Cmd_PosJog := FALSE;
   Chain3Long.Drive.Man.Cmd_NegJog := FALSE;
   Chain3Long.Drive.Man.Cmd_Step := FALSE;
   Chain3Long.Drive.Man.Cmd_Forward := FALSE;
   Chain3Long.Drive.Man.Cmd_Backward := FALSE;
   Chain3Long.Drive.Man.Cmd_Up := FALSE;
   Chain3Long.Drive.Man.Cmd_Down := FALSE;
   Chain3Long.Drive.Man.Cmd_Intermediate := FALSE;
   Chain3Long.Drive.Man.Cmd_Open := FALSE;
   Chain3Long.Drive.Man.Cmd_Close := FALSE;
   Chain3Long.Drive.Man.Cmd_PreOpen := FALSE;
   Chain3Long.Drive.Man.Cmd_Maintenance := FALSE;
   Chain3Long.Drive.Man.Cmd_OperatorSide := FALSE;
   Chain3Long.Drive.Man.Cmd_NotOperatorSide := FALSE;
   Chain3Long.Drive.Man.Cmd_OnMould := FALSE;
   Chain3Long.Drive.Man.Cmd_OffMould := FALSE;
   Chain3Long.Drive.Man.Cmd_Pos0 := FALSE;
   Chain3Long.Drive.Man.Cmd_Pos1 := FALSE;
   Chain3Long.Drive.Man.Cmd_Pos2 := FALSE;
   Chain3Long.Drive.Man.Cmd_Pos3 := FALSE;
   Chain3Long.Drive.Man.Cmd_Pos4 := FALSE;
   Chain3Long.Drive.Man.Cmd_Pos5 := FALSE;
   Chain3Long.Drive.Man.Ons_Step := FALSE;
   Chain3Long.Drive.Man.PhaseJogCmd := FALSE;
   Chain3Long.Drive.Man.CmdStartStep := FALSE;
   Chain3Long.Drive.Man.CmdEndStep := FALSE;
   Chain3Long.Drive.Man.StepCond := FALSE;
   Chain3Long.Drive.Man.TON_DelayHomeCmd.PT := T#3S;
   Chain3Long.Drive.Man.TON_DelayHomeCmd.IN := FALSE;
   Chain3Long.Drive.Auto.Cmd_Step := FALSE;
   Chain3Long.Drive.Auto.Cmd_StartStep := FALSE;
   Chain3Long.Drive.Auto.Cmd_EndStep := FALSE;
   Chain3Long.Drive.Auto.Cmd_Forward := FALSE;
   Chain3Long.Drive.Auto.Cmd_Backward := FALSE;
   Chain3Long.Drive.Auto.Cmd_Up := FALSE;
   Chain3Long.Drive.Auto.Cmd_Down := FALSE;
   Chain3Long.Drive.Auto.Cmd_Intermediate := FALSE;
   Chain3Long.Drive.Auto.Cmd_Open := FALSE;
   Chain3Long.Drive.Auto.Cmd_Close := FALSE;
   Chain3Long.Drive.Auto.Cmd_PreOpen := FALSE;
   Chain3Long.Drive.Auto.Cmd_Maintenance := FALSE;
   Chain3Long.Drive.Auto.Cmd_OperatorSide := FALSE;
   Chain3Long.Drive.Auto.Cmd_NotOperatorSide := FALSE;
   Chain3Long.Drive.Auto.Cmd_OnMould := FALSE;
   Chain3Long.Drive.Auto.Cmd_OffMould := FALSE;
   Chain3Long.Drive.Auto.Cmd_Pos0 := FALSE;
   Chain3Long.Drive.Auto.Cmd_Pos1 := FALSE;
   Chain3Long.Drive.Auto.Cmd_Pos2 := FALSE;
   Chain3Long.Drive.Auto.Cmd_Pos3 := FALSE;
   Chain3Long.Drive.Auto.Cmd_Pos4 := FALSE;
   Chain3Long.Drive.Auto.Cmd_Pos5 := FALSE;
   Chain3Long.Drive.Auto.Cmd_Gear := FALSE;
   Chain3Long.Drive.ACT.CMD.Enable := FALSE;
   Chain3Long.Drive.ACT.CMD.Pos_Mode := FALSE;
   Chain3Long.Drive.ACT.CMD.MergeDisabled := FALSE;
   Chain3Long.Drive.ACT.CMD.SCurve := FALSE;
   Chain3Long.Drive.ACT.CMD.Cam_Mode := TRUE;
   Chain3Long.Drive.ACT.CMD.Cam_Request := FALSE;
   Chain3Long.Drive.ACT.CMD.Cam_PhaseStop := FALSE;
   Chain3Long.Drive.ACT.CMD.Gear_Mode := FALSE;
   Chain3Long.Drive.ACT.CMD.Repos_Req := FALSE;
   Chain3Long.Drive.ACT.CMD.Jog_Pos := FALSE;
   Chain3Long.Drive.ACT.CMD.Jog_Neg := FALSE;
   Chain3Long.Drive.ACT.CMD.Stop := FALSE;
   Chain3Long.Drive.ACT.CMD.Calibration_Req := FALSE;
   Chain3Long.Drive.ACT.CMD.Reset := FALSE;
   Chain3Long.Drive.ACT.CMD.RegInput1 := FALSE;
   Chain3Long.Drive.ACT.CMD.Brake_Release := FALSE;
   Chain3Long.Drive.ACT.CMD.HwPosOvertravel_Dis := FALSE;
   Chain3Long.Drive.ACT.CMD.HwNegOvertravel_Dis := FALSE;
   Chain3Long.Drive.ACT.CMD.HwOvertravel_MSG_En := FALSE;
   Chain3Long.Drive.ACT.CMD.OneShootMove := FALSE;
   Chain3Long.Drive.ACT.CMD.Move_Type := 3;
   Chain3Long.Drive.ACT.CMD.Target_Pos := 0.0;
   Chain3Long.Drive.ACT.CMD.Speed := 0.0;
   Chain3Long.Drive.ACT.CMD.Acceleration := 300.0;
   Chain3Long.Drive.ACT.CMD.Deceleration := 300.0;
   Chain3Long.Drive.ACT.CMD.Torque_Limit := 30.0;
   Chain3Long.Drive.ACT.CMD.Gear_Ratio := 0.0;
   Chain3Long.Drive.ACT.CMD.Mccp_Length := 2;
   Chain3Long.Drive.ACT.CMD.Mccp_StartSlope := 0.0;
   Chain3Long.Drive.ACT.CMD.Mccp_EndSlope := 0.0;
   Chain3Long.Drive.ACT.CMD.Mapc_Direction := 1;
   Chain3Long.Drive.ACT.CMD.Mapc_SlaveScaling := 1.0;
   Chain3Long.Drive.ACT.CMD.Mapc_MasterScaling := 1.0;
   Chain3Long.Drive.ACT.CMD.Mapc_MasterLockPosition := 0.0;
   Chain3Long.Drive.ACT.CMD.Mapc_CamLockPosition := 0.0;
   Chain3Long.Drive.ACT.CMD.Cam[0].leadingValueStart := 0.0;
   Chain3Long.Drive.ACT.CMD.Cam[1].leadingValueStart := 162.0;
   Chain3Long.Drive.ACT.CMD.Cam[2..39].leadingValueStart := 0.0;
   Chain3Long.Drive.ACT.CMD.Cam[0].leadingValueEnd := 162.0;
   Chain3Long.Drive.ACT.CMD.Cam[1].leadingValueEnd := 360.0;
   Chain3Long.Drive.ACT.CMD.Cam[2..39].leadingValueEnd := 0.0;
   Chain3Long.Drive.ACT.CMD.Cam[0].followingValueStart := 0.0;
   Chain3Long.Drive.ACT.CMD.Cam[1].followingValueStart := 406.399993896484;
   Chain3Long.Drive.ACT.CMD.Cam[2..39].followingValueStart := 0.0;
   Chain3Long.Drive.ACT.CMD.Cam[0..1].followingValueEnd := 406.399993896484;
   Chain3Long.Drive.ACT.CMD.Cam[2..39].followingValueEnd := 0.0;
   Chain3Long.Drive.ACT.CMD.Cam[0..39].geoVeloStart := 0.0;
   Chain3Long.Drive.ACT.CMD.Cam[0..39].geoVeloEnd := 0.0;
   Chain3Long.Drive.ACT.CMD.Cam[0..39].geoAccelStart := 0.0;
   Chain3Long.Drive.ACT.CMD.Cam[0..39].geoAccelEnd := 0.0;
   Chain3Long.Drive.ACT.CMD.Cam[0..39].geoJerkStart := 0.0;
   Chain3Long.Drive.ACT.CMD.Cam[0..39].geoJerkEnd := 0.0;
   Chain3Long.Drive.ACT.CMD.Cam[0..39].inflectionPointParameter := 0.5;
   Chain3Long.Drive.ACT.CMD.Cam[0..39].modVeloTrapezoidParameter := 1.0;
   Chain3Long.Drive.ACT.CMD.Cam[0..39].modSineMaxAccelCaStar := 0.0;
   Chain3Long.Drive.ACT.CMD.Cam[0].camProfileType := 5;
   Chain3Long.Drive.ACT.CMD.Cam[1].camProfileType := 2;
   Chain3Long.Drive.ACT.CMD.Cam[2..39].camProfileType := 0;
   Chain3Long.Drive.ACT.FBK.Ready := TRUE;
   Chain3Long.Drive.ACT.FBK.Calibrated := TRUE;
   Chain3Long.Drive.ACT.FBK.Fault := FALSE;
   Chain3Long.Drive.ACT.FBK.ModuleConnFault := FALSE;
   Chain3Long.Drive.ACT.FBK.In_Position := FALSE;
   Chain3Long.Drive.ACT.FBK.Standstill := TRUE;
   Chain3Long.Drive.ACT.FBK.Enabled := FALSE;
   Chain3Long.Drive.ACT.FBK.BusReadyStatus := FALSE;
   Chain3Long.Drive.ACT.FBK.BrakeReleased := FALSE;
   Chain3Long.Drive.ACT.FBK.HwPosOvertravelDisabled := FALSE;
   Chain3Long.Drive.ACT.FBK.HwNegOvertravelDisabled := FALSE;
   Chain3Long.Drive.ACT.FBK.SafeOffStatus := FALSE;
   Chain3Long.Drive.ACT.FBK.MaxTorqueLimit := FALSE;
   Chain3Long.Drive.ACT.FBK.PosMerge_IP := FALSE;
   Chain3Long.Drive.ACT.FBK.PosMerge_PC := FALSE;
   Chain3Long.Drive.ACT.FBK.Gearing_IP := FALSE;
   Chain3Long.Drive.ACT.FBK.Position := 279.341;
   Chain3Long.Drive.ACT.FBK.Speed := 0.0;
   Chain3Long.Drive.ACT.FBK.Torque := 0.0;
   Chain3Long.Drive.ACT.FBK.RegInput1Pos := 0.0;
   Chain3Long.Drive.ACT.FBK.SeqCamErrorCode := 0;
   Chain3Long.Drive.ACT.FBK.SeqCamTargetPosMAM := 0.0;
   Chain3Long.Drive.ACT.FBK.SeqCamStatus.EndSequence := FALSE;
   Chain3Long.Drive.ACT.FBK.SeqCamStatus.EndSuccess := FALSE;
   Chain3Long.Drive.ACT.FBK.SeqCamStatus.EndError := FALSE;
   Chain3Long.Drive.ACT.FBK.SeqCamStatus.CamHook := FALSE;
   Chain3Long.Drive.ACT.FBK.SeqCamStatus.BothMapc_IP := FALSE;
   Chain3Long.Drive.ACT.FBK.SeqCamStatus.SlaveFwd := FALSE;
   Chain3Long.Drive.ACT.FBK.SeqCamStatus.SlaveBwd := FALSE;
   Chain3Long.Drive.ACT.FBK.SeqCamStatus.SlaveUnwind := FALSE;
   Chain3Long.Drive.ACT.FBK.SeqCamStatus.WaitValidByOpe := FALSE;
   Chain3Long.Drive.ACT.FBK.SeqCamStatus.MapcA_IP := FALSE;
   Chain3Long.Drive.ACT.FBK.SeqCamStatus.MapcB_IP := FALSE;
   Chain3Long.Drive.ACT.FBK.SeqCamStatus.MapcC_IP := FALSE;
   Chain3Long.Drive.ACT.FBK.SeqCamStatus.CamOnce_PC := FALSE;
   Chain3Long.Drive.ACT.FBK.SeqCamStatus.MaxDevError := FALSE;
   Chain3Long.Drive.ACT.FBK.SeqCamStatus.PositionCamLockStatus := FALSE;
   Chain3Long.Drive.ACT.FBK.SeqCamStatus.WaitRestart := FALSE;
   Chain3Long.Drive.ACT.FBK.SeqCamStatus.Bit17 := FALSE;
   Chain3Long.Drive.ACT.FBK.SeqCamStatus.Bit18 := FALSE;
   Chain3Long.Drive.ACT.FBK.SeqCamStatus.Bit19 := FALSE;
   Chain3Long.Drive.ACT.FBK.SeqCamStatus.Bit20 := FALSE;
   Chain3Long.Drive.ACT.FBK.SeqCamStatus.Bit21 := FALSE;
   Chain3Long.Drive.ACT.FBK.SeqCamStatus.Bit22 := FALSE;
   Chain3Long.Drive.ACT.FBK.SeqCamStatus.Bit23 := FALSE;
   Chain3Long.Drive.ACT.FBK.SeqCamStatus.Bit24 := FALSE;
   Chain3Long.Drive.ACT.FBK.SeqCamStatus.Bit25 := FALSE;
   Chain3Long.Drive.ACT.FBK.SeqCamStatus.Bit26 := FALSE;
   Chain3Long.Drive.ACT.FBK.SeqCamStatus.Bit27 := FALSE;
   Chain3Long.Drive.ACT.FBK.SeqCamStatus.Bit28 := FALSE;
   Chain3Long.Drive.ACT.FBK.SeqCamStatus.Bit29 := FALSE;
   Chain3Long.Drive.ACT.FBK.SeqCamStatus.Bit30 := FALSE;
   Chain3Long.Drive.ACT.FBK.SeqCamStatus.Bit31 := FALSE;
   Chain3Long.Drive.ACT.FBK.SeqCamStatus.Bit32 := FALSE;
   Chain3Long.Drive.PLS.FinePosOk.LowLimit := 405.4;
   Chain3Long.Drive.PLS.FinePosOk.HighLimit := 1.0;
   Chain3Long.Drive.PLS.FinePosOk.Ok := FALSE;
   Chain3Long.Drive.PLS.KeepPosOk.LowLimit := 404.4;
   Chain3Long.Drive.PLS.KeepPosOk.HighLimit := 2.0;
   Chain3Long.Drive.PLS.KeepPosOk.Ok := FALSE;
   Chain3Long.Drive.PLS.Up.LowLimit := 0.0;
   Chain3Long.Drive.PLS.Up.HighLimit := 0.0;
   Chain3Long.Drive.PLS.Up.Ok := FALSE;
   Chain3Long.Drive.PLS.Intermediate.LowLimit := 0.0;
   Chain3Long.Drive.PLS.Intermediate.HighLimit := 0.0;
   Chain3Long.Drive.PLS.Intermediate.Ok := FALSE;
   Chain3Long.Drive.PLS.Down.LowLimit := 0.0;
   Chain3Long.Drive.PLS.Down.HighLimit := 0.0;
   Chain3Long.Drive.PLS.Down.Ok := FALSE;
   Chain3Long.Drive.PLS.Forward.LowLimit := 0.0;
   Chain3Long.Drive.PLS.Forward.HighLimit := 0.0;
   Chain3Long.Drive.PLS.Forward.Ok := FALSE;
   Chain3Long.Drive.PLS.Backward.LowLimit := 0.0;
   Chain3Long.Drive.PLS.Backward.HighLimit := 0.0;
   Chain3Long.Drive.PLS.Backward.Ok := FALSE;
   Chain3Long.Drive.PLS.Open.LowLimit := 0.0;
   Chain3Long.Drive.PLS.Open.HighLimit := 0.0;
   Chain3Long.Drive.PLS.Open.Ok := FALSE;
   Chain3Long.Drive.PLS.Close.LowLimit := 0.0;
   Chain3Long.Drive.PLS.Close.HighLimit := 0.0;
   Chain3Long.Drive.PLS.Close.Ok := FALSE;
   Chain3Long.Drive.PLS.PreOpen.LowLimit := 0.0;
   Chain3Long.Drive.PLS.PreOpen.HighLimit := 0.0;
   Chain3Long.Drive.PLS.PreOpen.Ok := FALSE;
   Chain3Long.Drive.PLS.Maintenance.LowLimit := 0.0;
   Chain3Long.Drive.PLS.Maintenance.HighLimit := 0.0;
   Chain3Long.Drive.PLS.Maintenance.Ok := FALSE;
   Chain3Long.Drive.PLS.OperatorSide.LowLimit := 0.0;
   Chain3Long.Drive.PLS.OperatorSide.HighLimit := 0.0;
   Chain3Long.Drive.PLS.OperatorSide.Ok := FALSE;
   Chain3Long.Drive.PLS.NotOperatorSide.LowLimit := 0.0;
   Chain3Long.Drive.PLS.NotOperatorSide.HighLimit := 0.0;
   Chain3Long.Drive.PLS.NotOperatorSide.Ok := FALSE;
   Chain3Long.Drive.PLS.OnMould.LowLimit := 0.0;
   Chain3Long.Drive.PLS.OnMould.HighLimit := 0.0;
   Chain3Long.Drive.PLS.OnMould.Ok := FALSE;
   Chain3Long.Drive.PLS.OffMould.LowLimit := 0.0;
   Chain3Long.Drive.PLS.OffMould.HighLimit := 0.0;
   Chain3Long.Drive.PLS.OffMould.Ok := FALSE;
   Chain3Long.Drive.PLS.Pos0.LowLimit := 0.0;
   Chain3Long.Drive.PLS.Pos0.HighLimit := 0.0;
   Chain3Long.Drive.PLS.Pos0.Ok := FALSE;
   Chain3Long.Drive.PLS.Pos1.LowLimit := 0.0;
   Chain3Long.Drive.PLS.Pos1.HighLimit := 0.0;
   Chain3Long.Drive.PLS.Pos1.Ok := FALSE;
   Chain3Long.Drive.PLS.Pos2.LowLimit := 0.0;
   Chain3Long.Drive.PLS.Pos2.HighLimit := 0.0;
   Chain3Long.Drive.PLS.Pos2.Ok := FALSE;
   Chain3Long.Drive.PLS.Pos3.LowLimit := 0.0;
   Chain3Long.Drive.PLS.Pos3.HighLimit := 0.0;
   Chain3Long.Drive.PLS.Pos3.Ok := FALSE;
   Chain3Long.Drive.PLS.Pos4.LowLimit := 0.0;
   Chain3Long.Drive.PLS.Pos4.HighLimit := 0.0;
   Chain3Long.Drive.PLS.Pos4.Ok := FALSE;
   Chain3Long.Drive.PLS.Pos5.LowLimit := 0.0;
   Chain3Long.Drive.PLS.Pos5.HighLimit := 0.0;
   Chain3Long.Drive.PLS.Pos5.Ok := FALSE;
   Chain3Long.Drive.TON_EnableDrive.PT := T#500MS;
   Chain3Long.Drive.TON_EnableDrive.IN := FALSE;
   Chain3Long.Drive.TON_HwOvertravel_Dis.PT := T#0MS;
   Chain3Long.Drive.TON_HwOvertravel_Dis.IN := FALSE;
   Chain3Long.Drive.TON_HwOvertravel_En.PT := T#0MS;
   Chain3Long.Drive.TON_HwOvertravel_En.IN := FALSE;
   Chain3Long.Drive.TON_TimeoutMovement.PT := T#0MS;
   Chain3Long.Drive.TON_TimeoutMovement.IN := FALSE;
   Chain4Cross.AlmOk := TRUE;
   Chain4Cross.StationWorked := TRUE;
   Chain4Cross.CheckObstruction := FALSE;
   Chain4Cross.OutChainObstruction := TRUE;
   Chain4Cross.StrobeWork := FALSE;
   Chain4Cross.StrobeShift := FALSE;
   Chain4Cross.ManualMovement := FALSE;
   Chain4Cross.OkToStop := TRUE;
   Chain4Cross.PosOk := TRUE;
   Chain4Cross.Ons_PosOk := TRUE;
   Chain4Cross.EnaMove := TRUE;
   Chain4Cross.StationEna := TRUE;
   Chain4Cross.ModeLong := FALSE;
   Chain4Cross.ModeCross := TRUE;
   Chain4Cross.ModeCont := FALSE;
   Chain4Cross.Cfg_Mould_ChainSteps := 1;
   Chain4Cross.Cfg_Mould_EndPos := 7;
   Chain4Cross.Shift_Lenght := 8;
   Chain4Cross.PosMasterAdvanceStep := 0.0;
   Chain4Cross.Input.EndChaMouPre := FALSE;
   Chain4Cross.Input.PshHig := FALSE;
   Chain4Cross.Input.PshLow := FALSE;
   Chain4Cross.Output.PshHig := FALSE;
   Chain4Cross.Output.PshLow := FALSE;
   Chain4Cross.Man.EnaPbt := FALSE;
   Chain4Cross.Man.RstCmd := TRUE;
   Chain4Cross.Man.ScreenNumber := 300_040_301;
   Chain4Cross.Man.WithinScreenRange := 0;
   Chain4Cross.Drive.AlmOk := FALSE;
   Chain4Cross.Drive.AlmEmerg := FALSE;
   Chain4Cross.Drive.AlmNode := FALSE;
   Chain4Cross.Drive.InitPosDrive := FALSE;
   Chain4Cross.Drive.InitPosDrivePLS := FALSE;
   Chain4Cross.Drive.GearingON := FALSE;
   Chain4Cross.Drive.CamHook := FALSE;
   Chain4Cross.Drive.CamStoppingPhase := FALSE;
   Chain4Cross.Drive.RepositioningRequest := FALSE;
   Chain4Cross.Drive.CamRequestResult := FALSE;
   Chain4Cross.Drive.CamRequestError := FALSE;
   Chain4Cross.Drive.CamRequestOk := TRUE;
   Chain4Cross.Drive.CalibDisAxisReq := FALSE;
   Chain4Cross.Drive.CalibReq := FALSE;
   Chain4Cross.Drive.CalibProcess := FALSE;
   Chain4Cross.Drive.HwOvertravelDisReq := FALSE;
   Chain4Cross.Drive.HwOvertravelEnReq := FALSE;
   Chain4Cross.Drive.AuxCamRequest := FALSE;
   Chain4Cross.Drive.TorquePeakEna := TRUE;
   Chain4Cross.Drive.Cmd_Repos := FALSE;
   Chain4Cross.Drive.Ons_CamRequest := FALSE;
   Chain4Cross.Drive.AuxCmdPosition := 0;
   Chain4Cross.Drive.Unwind := 812.8;
   Chain4Cross.Drive.MaxDev := 150.0;
   Chain4Cross.Drive.ReposSpeed := 10.0;
   Chain4Cross.Drive.CalcSlaveDifferenceABS := 0.0;
   Chain4Cross.Drive.CalcModPosition := 0.0;
   Chain4Cross.Drive.CalcSlaveDifference := 0.0;
   Chain4Cross.Drive.CalcMinDeltaPos := 0.0;
   Chain4Cross.Drive.CalcMaxDeltaPos := 0.0;
   Chain4Cross.Drive.CalcHalfPosUnwind := 0.0;
   Chain4Cross.Drive.Man.Cmd_PosJog := FALSE;
   Chain4Cross.Drive.Man.Cmd_NegJog := FALSE;
   Chain4Cross.Drive.Man.Cmd_Step := FALSE;
   Chain4Cross.Drive.Man.Cmd_Forward := FALSE;
   Chain4Cross.Drive.Man.Cmd_Backward := FALSE;
   Chain4Cross.Drive.Man.Cmd_Up := FALSE;
   Chain4Cross.Drive.Man.Cmd_Down := FALSE;
   Chain4Cross.Drive.Man.Cmd_Intermediate := FALSE;
   Chain4Cross.Drive.Man.Cmd_Open := FALSE;
   Chain4Cross.Drive.Man.Cmd_Close := FALSE;
   Chain4Cross.Drive.Man.Cmd_PreOpen := FALSE;
   Chain4Cross.Drive.Man.Cmd_Maintenance := FALSE;
   Chain4Cross.Drive.Man.Cmd_OperatorSide := FALSE;
   Chain4Cross.Drive.Man.Cmd_NotOperatorSide := FALSE;
   Chain4Cross.Drive.Man.Cmd_OnMould := FALSE;
   Chain4Cross.Drive.Man.Cmd_OffMould := FALSE;
   Chain4Cross.Drive.Man.Cmd_Pos0 := FALSE;
   Chain4Cross.Drive.Man.Cmd_Pos1 := FALSE;
   Chain4Cross.Drive.Man.Cmd_Pos2 := FALSE;
   Chain4Cross.Drive.Man.Cmd_Pos3 := FALSE;
   Chain4Cross.Drive.Man.Cmd_Pos4 := FALSE;
   Chain4Cross.Drive.Man.Cmd_Pos5 := FALSE;
   Chain4Cross.Drive.Man.Ons_Step := FALSE;
   Chain4Cross.Drive.Man.PhaseJogCmd := TRUE;
   Chain4Cross.Drive.Man.CmdStartStep := FALSE;
   Chain4Cross.Drive.Man.CmdEndStep := FALSE;
   Chain4Cross.Drive.Man.StepCond := FALSE;
   Chain4Cross.Drive.Man.TON_DelayHomeCmd.PT := T#3S;
   Chain4Cross.Drive.Man.TON_DelayHomeCmd.IN := FALSE;
   Chain4Cross.Drive.Auto.Cmd_Step := FALSE;
   Chain4Cross.Drive.Auto.Cmd_StartStep := FALSE;
   Chain4Cross.Drive.Auto.Cmd_EndStep := FALSE;
   Chain4Cross.Drive.Auto.Cmd_Forward := FALSE;
   Chain4Cross.Drive.Auto.Cmd_Backward := FALSE;
   Chain4Cross.Drive.Auto.Cmd_Up := FALSE;
   Chain4Cross.Drive.Auto.Cmd_Down := FALSE;
   Chain4Cross.Drive.Auto.Cmd_Intermediate := FALSE;
   Chain4Cross.Drive.Auto.Cmd_Open := FALSE;
   Chain4Cross.Drive.Auto.Cmd_Close := FALSE;
   Chain4Cross.Drive.Auto.Cmd_PreOpen := FALSE;
   Chain4Cross.Drive.Auto.Cmd_Maintenance := FALSE;
   Chain4Cross.Drive.Auto.Cmd_OperatorSide := FALSE;
   Chain4Cross.Drive.Auto.Cmd_NotOperatorSide := FALSE;
   Chain4Cross.Drive.Auto.Cmd_OnMould := FALSE;
   Chain4Cross.Drive.Auto.Cmd_OffMould := FALSE;
   Chain4Cross.Drive.Auto.Cmd_Pos0 := FALSE;
   Chain4Cross.Drive.Auto.Cmd_Pos1 := FALSE;
   Chain4Cross.Drive.Auto.Cmd_Pos2 := FALSE;
   Chain4Cross.Drive.Auto.Cmd_Pos3 := FALSE;
   Chain4Cross.Drive.Auto.Cmd_Pos4 := FALSE;
   Chain4Cross.Drive.Auto.Cmd_Pos5 := FALSE;
   Chain4Cross.Drive.Auto.Cmd_Gear := FALSE;
   Chain4Cross.Drive.ACT.CMD.Enable := FALSE;
   Chain4Cross.Drive.ACT.CMD.Pos_Mode := FALSE;
   Chain4Cross.Drive.ACT.CMD.MergeDisabled := FALSE;
   Chain4Cross.Drive.ACT.CMD.SCurve := FALSE;
   Chain4Cross.Drive.ACT.CMD.Cam_Mode := TRUE;
   Chain4Cross.Drive.ACT.CMD.Cam_Request := FALSE;
   Chain4Cross.Drive.ACT.CMD.Cam_PhaseStop := FALSE;
   Chain4Cross.Drive.ACT.CMD.Gear_Mode := FALSE;
   Chain4Cross.Drive.ACT.CMD.Repos_Req := FALSE;
   Chain4Cross.Drive.ACT.CMD.Jog_Pos := FALSE;
   Chain4Cross.Drive.ACT.CMD.Jog_Neg := FALSE;
   Chain4Cross.Drive.ACT.CMD.Stop := FALSE;
   Chain4Cross.Drive.ACT.CMD.Calibration_Req := FALSE;
   Chain4Cross.Drive.ACT.CMD.Reset := FALSE;
   Chain4Cross.Drive.ACT.CMD.RegInput1 := FALSE;
   Chain4Cross.Drive.ACT.CMD.Brake_Release := FALSE;
   Chain4Cross.Drive.ACT.CMD.HwPosOvertravel_Dis := FALSE;
   Chain4Cross.Drive.ACT.CMD.HwNegOvertravel_Dis := FALSE;
   Chain4Cross.Drive.ACT.CMD.HwOvertravel_MSG_En := FALSE;
   Chain4Cross.Drive.ACT.CMD.OneShootMove := FALSE;
   Chain4Cross.Drive.ACT.CMD.Move_Type := 3;
   Chain4Cross.Drive.ACT.CMD.Target_Pos := 0.0;
   Chain4Cross.Drive.ACT.CMD.Speed := 0.0;
   Chain4Cross.Drive.ACT.CMD.Acceleration := 300.0;
   Chain4Cross.Drive.ACT.CMD.Deceleration := 300.0;
   Chain4Cross.Drive.ACT.CMD.Torque_Limit := 30.0;
   Chain4Cross.Drive.ACT.CMD.Gear_Ratio := 0.0;
   Chain4Cross.Drive.ACT.CMD.Mccp_Length := 6;
   Chain4Cross.Drive.ACT.CMD.Mccp_StartSlope := 0.0;
   Chain4Cross.Drive.ACT.CMD.Mccp_EndSlope := 0.0;
   Chain4Cross.Drive.ACT.CMD.Mapc_Direction := 1;
   Chain4Cross.Drive.ACT.CMD.Mapc_SlaveScaling := 1.0;
   Chain4Cross.Drive.ACT.CMD.Mapc_MasterScaling := 1.0;
   Chain4Cross.Drive.ACT.CMD.Mapc_MasterLockPosition := 0.0;
   Chain4Cross.Drive.ACT.CMD.Mapc_CamLockPosition := 0.0;
   Chain4Cross.Drive.ACT.CMD.Cam[0].leadingValueStart := 0.0;
   Chain4Cross.Drive.ACT.CMD.Cam[1].leadingValueStart := 193.679992675781;
   Chain4Cross.Drive.ACT.CMD.Cam[2..3].leadingValueStart := 225.360000610352;
   Chain4Cross.Drive.ACT.CMD.Cam[4].leadingValueStart := 328.320007324219;
   Chain4Cross.Drive.ACT.CMD.Cam[5].leadingValueStart := 360.0;
   Chain4Cross.Drive.ACT.CMD.Cam[6..39].leadingValueStart := 0.0;
   Chain4Cross.Drive.ACT.CMD.Cam[0].leadingValueEnd := 162.0;
   Chain4Cross.Drive.ACT.CMD.Cam[1..2].leadingValueEnd := 0.0;
   Chain4Cross.Drive.ACT.CMD.Cam[3].leadingValueEnd := 296.640014648438;
   Chain4Cross.Drive.ACT.CMD.Cam[4..39].leadingValueEnd := 0.0;
   Chain4Cross.Drive.ACT.CMD.Cam[0].followingValueStart := 0.0;
   Chain4Cross.Drive.ACT.CMD.Cam[1].followingValueStart := 31.8745098114014;
   Chain4Cross.Drive.ACT.CMD.Cam[2..3].followingValueStart := 191.247055053711;
   Chain4Cross.Drive.ACT.CMD.Cam[4].followingValueStart := 780.925476074219;
   Chain4Cross.Drive.ACT.CMD.Cam[5].followingValueStart := 812.799987792969;
   Chain4Cross.Drive.ACT.CMD.Cam[6..39].followingValueStart := 0.0;
   Chain4Cross.Drive.ACT.CMD.Cam[0..2].followingValueEnd := 0.0;
   Chain4Cross.Drive.ACT.CMD.Cam[3].followingValueEnd := 621.552917480469;
   Chain4Cross.Drive.ACT.CMD.Cam[4..39].followingValueEnd := 0.0;
   Chain4Cross.Drive.ACT.CMD.Cam[0..39].geoVeloStart := 0.0;
   Chain4Cross.Drive.ACT.CMD.Cam[0..39].geoVeloEnd := 0.0;
   Chain4Cross.Drive.ACT.CMD.Cam[0..39].geoAccelStart := 0.0;
   Chain4Cross.Drive.ACT.CMD.Cam[0..39].geoAccelEnd := 0.0;
   Chain4Cross.Drive.ACT.CMD.Cam[0..39].geoJerkStart := 0.0;
   Chain4Cross.Drive.ACT.CMD.Cam[0..39].geoJerkEnd := 0.0;
   Chain4Cross.Drive.ACT.CMD.Cam[0..39].inflectionPointParameter := 0.5;
   Chain4Cross.Drive.ACT.CMD.Cam[0..39].modVeloTrapezoidParameter := 1.0;
   Chain4Cross.Drive.ACT.CMD.Cam[0..39].modSineMaxAccelCaStar := 0.0;
   Chain4Cross.Drive.ACT.CMD.Cam[0].camProfileType := 2;
   Chain4Cross.Drive.ACT.CMD.Cam[1..2].camProfileType := 1;
   Chain4Cross.Drive.ACT.CMD.Cam[3].camProfileType := 3;
   Chain4Cross.Drive.ACT.CMD.Cam[4..5].camProfileType := 1;
   Chain4Cross.Drive.ACT.CMD.Cam[6..39].camProfileType := 0;
   Chain4Cross.Drive.ACT.FBK.Ready := TRUE;
   Chain4Cross.Drive.ACT.FBK.Calibrated := TRUE;
   Chain4Cross.Drive.ACT.FBK.Fault := FALSE;
   Chain4Cross.Drive.ACT.FBK.ModuleConnFault := FALSE;
   Chain4Cross.Drive.ACT.FBK.In_Position := FALSE;
   Chain4Cross.Drive.ACT.FBK.Standstill := TRUE;
   Chain4Cross.Drive.ACT.FBK.Enabled := FALSE;
   Chain4Cross.Drive.ACT.FBK.BusReadyStatus := FALSE;
   Chain4Cross.Drive.ACT.FBK.BrakeReleased := FALSE;
   Chain4Cross.Drive.ACT.FBK.HwPosOvertravelDisabled := FALSE;
   Chain4Cross.Drive.ACT.FBK.HwNegOvertravelDisabled := FALSE;
   Chain4Cross.Drive.ACT.FBK.SafeOffStatus := FALSE;
   Chain4Cross.Drive.ACT.FBK.MaxTorqueLimit := FALSE;
   Chain4Cross.Drive.ACT.FBK.PosMerge_IP := FALSE;
   Chain4Cross.Drive.ACT.FBK.PosMerge_PC := FALSE;
   Chain4Cross.Drive.ACT.FBK.Gearing_IP := FALSE;
   Chain4Cross.Drive.ACT.FBK.Position := 0.099;
   Chain4Cross.Drive.ACT.FBK.Speed := 0.0;
   Chain4Cross.Drive.ACT.FBK.Torque := 0.0;
   Chain4Cross.Drive.ACT.FBK.RegInput1Pos := 0.0;
   Chain4Cross.Drive.ACT.FBK.SeqCamErrorCode := 0;
   Chain4Cross.Drive.ACT.FBK.SeqCamTargetPosMAM := 0.0;
   Chain4Cross.Drive.ACT.FBK.SeqCamStatus.EndSequence := FALSE;
   Chain4Cross.Drive.ACT.FBK.SeqCamStatus.EndSuccess := FALSE;
   Chain4Cross.Drive.ACT.FBK.SeqCamStatus.EndError := FALSE;
   Chain4Cross.Drive.ACT.FBK.SeqCamStatus.CamHook := FALSE;
   Chain4Cross.Drive.ACT.FBK.SeqCamStatus.BothMapc_IP := FALSE;
   Chain4Cross.Drive.ACT.FBK.SeqCamStatus.SlaveFwd := FALSE;
   Chain4Cross.Drive.ACT.FBK.SeqCamStatus.SlaveBwd := FALSE;
   Chain4Cross.Drive.ACT.FBK.SeqCamStatus.SlaveUnwind := FALSE;
   Chain4Cross.Drive.ACT.FBK.SeqCamStatus.WaitValidByOpe := FALSE;
   Chain4Cross.Drive.ACT.FBK.SeqCamStatus.MapcA_IP := FALSE;
   Chain4Cross.Drive.ACT.FBK.SeqCamStatus.MapcB_IP := FALSE;
   Chain4Cross.Drive.ACT.FBK.SeqCamStatus.MapcC_IP := FALSE;
   Chain4Cross.Drive.ACT.FBK.SeqCamStatus.CamOnce_PC := FALSE;
   Chain4Cross.Drive.ACT.FBK.SeqCamStatus.MaxDevError := FALSE;
   Chain4Cross.Drive.ACT.FBK.SeqCamStatus.PositionCamLockStatus := FALSE;
   Chain4Cross.Drive.ACT.FBK.SeqCamStatus.WaitRestart := FALSE;
   Chain4Cross.Drive.ACT.FBK.SeqCamStatus.Bit17 := FALSE;
   Chain4Cross.Drive.ACT.FBK.SeqCamStatus.Bit18 := FALSE;
   Chain4Cross.Drive.ACT.FBK.SeqCamStatus.Bit19 := FALSE;
   Chain4Cross.Drive.ACT.FBK.SeqCamStatus.Bit20 := FALSE;
   Chain4Cross.Drive.ACT.FBK.SeqCamStatus.Bit21 := FALSE;
   Chain4Cross.Drive.ACT.FBK.SeqCamStatus.Bit22 := FALSE;
   Chain4Cross.Drive.ACT.FBK.SeqCamStatus.Bit23 := FALSE;
   Chain4Cross.Drive.ACT.FBK.SeqCamStatus.Bit24 := FALSE;
   Chain4Cross.Drive.ACT.FBK.SeqCamStatus.Bit25 := FALSE;
   Chain4Cross.Drive.ACT.FBK.SeqCamStatus.Bit26 := FALSE;
   Chain4Cross.Drive.ACT.FBK.SeqCamStatus.Bit27 := FALSE;
   Chain4Cross.Drive.ACT.FBK.SeqCamStatus.Bit28 := FALSE;
   Chain4Cross.Drive.ACT.FBK.SeqCamStatus.Bit29 := FALSE;
   Chain4Cross.Drive.ACT.FBK.SeqCamStatus.Bit30 := FALSE;
   Chain4Cross.Drive.ACT.FBK.SeqCamStatus.Bit31 := FALSE;
   Chain4Cross.Drive.ACT.FBK.SeqCamStatus.Bit32 := FALSE;
   Chain4Cross.Drive.PLS.FinePosOk.LowLimit := 811.8;
   Chain4Cross.Drive.PLS.FinePosOk.HighLimit := 1.0;
   Chain4Cross.Drive.PLS.FinePosOk.Ok := TRUE;
   Chain4Cross.Drive.PLS.KeepPosOk.LowLimit := 810.8;
   Chain4Cross.Drive.PLS.KeepPosOk.HighLimit := 2.0;
   Chain4Cross.Drive.PLS.KeepPosOk.Ok := TRUE;
   Chain4Cross.Drive.PLS.Up.LowLimit := 0.0;
   Chain4Cross.Drive.PLS.Up.HighLimit := 0.0;
   Chain4Cross.Drive.PLS.Up.Ok := FALSE;
   Chain4Cross.Drive.PLS.Intermediate.LowLimit := 0.0;
   Chain4Cross.Drive.PLS.Intermediate.HighLimit := 0.0;
   Chain4Cross.Drive.PLS.Intermediate.Ok := FALSE;
   Chain4Cross.Drive.PLS.Down.LowLimit := 0.0;
   Chain4Cross.Drive.PLS.Down.HighLimit := 0.0;
   Chain4Cross.Drive.PLS.Down.Ok := FALSE;
   Chain4Cross.Drive.PLS.Forward.LowLimit := 0.0;
   Chain4Cross.Drive.PLS.Forward.HighLimit := 0.0;
   Chain4Cross.Drive.PLS.Forward.Ok := FALSE;
   Chain4Cross.Drive.PLS.Backward.LowLimit := 0.0;
   Chain4Cross.Drive.PLS.Backward.HighLimit := 0.0;
   Chain4Cross.Drive.PLS.Backward.Ok := FALSE;
   Chain4Cross.Drive.PLS.Open.LowLimit := 0.0;
   Chain4Cross.Drive.PLS.Open.HighLimit := 0.0;
   Chain4Cross.Drive.PLS.Open.Ok := FALSE;
   Chain4Cross.Drive.PLS.Close.LowLimit := 0.0;
   Chain4Cross.Drive.PLS.Close.HighLimit := 0.0;
   Chain4Cross.Drive.PLS.Close.Ok := FALSE;
   Chain4Cross.Drive.PLS.PreOpen.LowLimit := 0.0;
   Chain4Cross.Drive.PLS.PreOpen.HighLimit := 0.0;
   Chain4Cross.Drive.PLS.PreOpen.Ok := FALSE;
   Chain4Cross.Drive.PLS.Maintenance.LowLimit := 0.0;
   Chain4Cross.Drive.PLS.Maintenance.HighLimit := 0.0;
   Chain4Cross.Drive.PLS.Maintenance.Ok := FALSE;
   Chain4Cross.Drive.PLS.OperatorSide.LowLimit := 0.0;
   Chain4Cross.Drive.PLS.OperatorSide.HighLimit := 0.0;
   Chain4Cross.Drive.PLS.OperatorSide.Ok := FALSE;
   Chain4Cross.Drive.PLS.NotOperatorSide.LowLimit := 0.0;
   Chain4Cross.Drive.PLS.NotOperatorSide.HighLimit := 0.0;
   Chain4Cross.Drive.PLS.NotOperatorSide.Ok := FALSE;
   Chain4Cross.Drive.PLS.OnMould.LowLimit := 0.0;
   Chain4Cross.Drive.PLS.OnMould.HighLimit := 0.0;
   Chain4Cross.Drive.PLS.OnMould.Ok := FALSE;
   Chain4Cross.Drive.PLS.OffMould.LowLimit := 0.0;
   Chain4Cross.Drive.PLS.OffMould.HighLimit := 0.0;
   Chain4Cross.Drive.PLS.OffMould.Ok := FALSE;
   Chain4Cross.Drive.PLS.Pos0.LowLimit := 0.0;
   Chain4Cross.Drive.PLS.Pos0.HighLimit := 0.0;
   Chain4Cross.Drive.PLS.Pos0.Ok := FALSE;
   Chain4Cross.Drive.PLS.Pos1.LowLimit := 0.0;
   Chain4Cross.Drive.PLS.Pos1.HighLimit := 0.0;
   Chain4Cross.Drive.PLS.Pos1.Ok := FALSE;
   Chain4Cross.Drive.PLS.Pos2.LowLimit := 0.0;
   Chain4Cross.Drive.PLS.Pos2.HighLimit := 0.0;
   Chain4Cross.Drive.PLS.Pos2.Ok := FALSE;
   Chain4Cross.Drive.PLS.Pos3.LowLimit := 0.0;
   Chain4Cross.Drive.PLS.Pos3.HighLimit := 0.0;
   Chain4Cross.Drive.PLS.Pos3.Ok := FALSE;
   Chain4Cross.Drive.PLS.Pos4.LowLimit := 0.0;
   Chain4Cross.Drive.PLS.Pos4.HighLimit := 0.0;
   Chain4Cross.Drive.PLS.Pos4.Ok := FALSE;
   Chain4Cross.Drive.PLS.Pos5.LowLimit := 0.0;
   Chain4Cross.Drive.PLS.Pos5.HighLimit := 0.0;
   Chain4Cross.Drive.PLS.Pos5.Ok := FALSE;
   Chain4Cross.Drive.TON_EnableDrive.PT := T#500MS;
   Chain4Cross.Drive.TON_EnableDrive.IN := FALSE;
   Chain4Cross.Drive.TON_HwOvertravel_Dis.PT := T#0MS;
   Chain4Cross.Drive.TON_HwOvertravel_Dis.IN := FALSE;
   Chain4Cross.Drive.TON_HwOvertravel_En.PT := T#0MS;
   Chain4Cross.Drive.TON_HwOvertravel_En.IN := FALSE;
   Chain4Cross.Drive.TON_TimeoutMovement.PT := T#0MS;
   Chain4Cross.Drive.TON_TimeoutMovement.IN := FALSE;
   Chain5Long.AlmOk := TRUE;
   Chain5Long.StationWorked := TRUE;
   Chain5Long.CheckObstruction := TRUE;
   Chain5Long.OutChainObstruction := TRUE;
   Chain5Long.StrobeWork := FALSE;
   Chain5Long.StrobeShift := FALSE;
   Chain5Long.ManualMovement := FALSE;
   Chain5Long.OkToStop := TRUE;
   Chain5Long.PosOk := FALSE;
   Chain5Long.Ons_PosOk := FALSE;
   Chain5Long.EnaMove := TRUE;
   Chain5Long.StationEna := FALSE;
   Chain5Long.ModeLong := TRUE;
   Chain5Long.ModeCross := FALSE;
   Chain5Long.ModeCont := FALSE;
   Chain5Long.Cfg_Mould_ChainSteps := 1;
   Chain5Long.Cfg_Mould_EndPos := 88;
   Chain5Long.Shift_Lenght := 89;
   Chain5Long.PosMasterAdvanceStep := 0.0;
   Chain5Long.Input.EndChaMouPre := FALSE;
   Chain5Long.Input.PshHig := FALSE;
   Chain5Long.Input.PshLow := FALSE;
   Chain5Long.Output.PshHig := FALSE;
   Chain5Long.Output.PshLow := FALSE;
   Chain5Long.Man.EnaPbt := FALSE;
   Chain5Long.Man.RstCmd := TRUE;
   Chain5Long.Man.ScreenNumber := 300_050_301;
   Chain5Long.Man.WithinScreenRange := 0;
   Chain5Long.Drive.AlmOk := FALSE;
   Chain5Long.Drive.AlmEmerg := FALSE;
   Chain5Long.Drive.AlmNode := FALSE;
   Chain5Long.Drive.InitPosDrive := FALSE;
   Chain5Long.Drive.InitPosDrivePLS := FALSE;
   Chain5Long.Drive.GearingON := FALSE;
   Chain5Long.Drive.CamHook := FALSE;
   Chain5Long.Drive.CamStoppingPhase := FALSE;
   Chain5Long.Drive.RepositioningRequest := FALSE;
   Chain5Long.Drive.CamRequestResult := FALSE;
   Chain5Long.Drive.CamRequestError := FALSE;
   Chain5Long.Drive.CamRequestOk := TRUE;
   Chain5Long.Drive.CalibDisAxisReq := FALSE;
   Chain5Long.Drive.CalibReq := FALSE;
   Chain5Long.Drive.CalibProcess := FALSE;
   Chain5Long.Drive.HwOvertravelDisReq := FALSE;
   Chain5Long.Drive.HwOvertravelEnReq := FALSE;
   Chain5Long.Drive.AuxCamRequest := FALSE;
   Chain5Long.Drive.TorquePeakEna := TRUE;
   Chain5Long.Drive.Cmd_Repos := FALSE;
   Chain5Long.Drive.Ons_CamRequest := FALSE;
   Chain5Long.Drive.AuxCmdPosition := 0;
   Chain5Long.Drive.Unwind := 406.4;
   Chain5Long.Drive.MaxDev := 150.0;
   Chain5Long.Drive.ReposSpeed := 10.0;
   Chain5Long.Drive.CalcSlaveDifferenceABS := 0.0;
   Chain5Long.Drive.CalcModPosition := 0.0;
   Chain5Long.Drive.CalcSlaveDifference := 0.0;
   Chain5Long.Drive.CalcMinDeltaPos := 0.0;
   Chain5Long.Drive.CalcMaxDeltaPos := 0.0;
   Chain5Long.Drive.CalcHalfPosUnwind := 0.0;
   Chain5Long.Drive.Man.Cmd_PosJog := FALSE;
   Chain5Long.Drive.Man.Cmd_NegJog := FALSE;
   Chain5Long.Drive.Man.Cmd_Step := FALSE;
   Chain5Long.Drive.Man.Cmd_Forward := FALSE;
   Chain5Long.Drive.Man.Cmd_Backward := FALSE;
   Chain5Long.Drive.Man.Cmd_Up := FALSE;
   Chain5Long.Drive.Man.Cmd_Down := FALSE;
   Chain5Long.Drive.Man.Cmd_Intermediate := FALSE;
   Chain5Long.Drive.Man.Cmd_Open := FALSE;
   Chain5Long.Drive.Man.Cmd_Close := FALSE;
   Chain5Long.Drive.Man.Cmd_PreOpen := FALSE;
   Chain5Long.Drive.Man.Cmd_Maintenance := FALSE;
   Chain5Long.Drive.Man.Cmd_OperatorSide := FALSE;
   Chain5Long.Drive.Man.Cmd_NotOperatorSide := FALSE;
   Chain5Long.Drive.Man.Cmd_OnMould := FALSE;
   Chain5Long.Drive.Man.Cmd_OffMould := FALSE;
   Chain5Long.Drive.Man.Cmd_Pos0 := FALSE;
   Chain5Long.Drive.Man.Cmd_Pos1 := FALSE;
   Chain5Long.Drive.Man.Cmd_Pos2 := FALSE;
   Chain5Long.Drive.Man.Cmd_Pos3 := FALSE;
   Chain5Long.Drive.Man.Cmd_Pos4 := FALSE;
   Chain5Long.Drive.Man.Cmd_Pos5 := FALSE;
   Chain5Long.Drive.Man.Ons_Step := FALSE;
   Chain5Long.Drive.Man.PhaseJogCmd := FALSE;
   Chain5Long.Drive.Man.CmdStartStep := FALSE;
   Chain5Long.Drive.Man.CmdEndStep := FALSE;
   Chain5Long.Drive.Man.StepCond := FALSE;
   Chain5Long.Drive.Man.TON_DelayHomeCmd.PT := T#3S;
   Chain5Long.Drive.Man.TON_DelayHomeCmd.IN := FALSE;
   Chain5Long.Drive.Auto.Cmd_Step := FALSE;
   Chain5Long.Drive.Auto.Cmd_StartStep := FALSE;
   Chain5Long.Drive.Auto.Cmd_EndStep := FALSE;
   Chain5Long.Drive.Auto.Cmd_Forward := FALSE;
   Chain5Long.Drive.Auto.Cmd_Backward := FALSE;
   Chain5Long.Drive.Auto.Cmd_Up := FALSE;
   Chain5Long.Drive.Auto.Cmd_Down := FALSE;
   Chain5Long.Drive.Auto.Cmd_Intermediate := FALSE;
   Chain5Long.Drive.Auto.Cmd_Open := FALSE;
   Chain5Long.Drive.Auto.Cmd_Close := FALSE;
   Chain5Long.Drive.Auto.Cmd_PreOpen := FALSE;
   Chain5Long.Drive.Auto.Cmd_Maintenance := FALSE;
   Chain5Long.Drive.Auto.Cmd_OperatorSide := FALSE;
   Chain5Long.Drive.Auto.Cmd_NotOperatorSide := FALSE;
   Chain5Long.Drive.Auto.Cmd_OnMould := FALSE;
   Chain5Long.Drive.Auto.Cmd_OffMould := FALSE;
   Chain5Long.Drive.Auto.Cmd_Pos0 := FALSE;
   Chain5Long.Drive.Auto.Cmd_Pos1 := FALSE;
   Chain5Long.Drive.Auto.Cmd_Pos2 := FALSE;
   Chain5Long.Drive.Auto.Cmd_Pos3 := FALSE;
   Chain5Long.Drive.Auto.Cmd_Pos4 := FALSE;
   Chain5Long.Drive.Auto.Cmd_Pos5 := FALSE;
   Chain5Long.Drive.Auto.Cmd_Gear := FALSE;
   Chain5Long.Drive.ACT.CMD.Enable := FALSE;
   Chain5Long.Drive.ACT.CMD.Pos_Mode := FALSE;
   Chain5Long.Drive.ACT.CMD.MergeDisabled := FALSE;
   Chain5Long.Drive.ACT.CMD.SCurve := FALSE;
   Chain5Long.Drive.ACT.CMD.Cam_Mode := TRUE;
   Chain5Long.Drive.ACT.CMD.Cam_Request := FALSE;
   Chain5Long.Drive.ACT.CMD.Cam_PhaseStop := FALSE;
   Chain5Long.Drive.ACT.CMD.Gear_Mode := FALSE;
   Chain5Long.Drive.ACT.CMD.Repos_Req := FALSE;
   Chain5Long.Drive.ACT.CMD.Jog_Pos := FALSE;
   Chain5Long.Drive.ACT.CMD.Jog_Neg := FALSE;
   Chain5Long.Drive.ACT.CMD.Stop := FALSE;
   Chain5Long.Drive.ACT.CMD.Calibration_Req := FALSE;
   Chain5Long.Drive.ACT.CMD.Reset := FALSE;
   Chain5Long.Drive.ACT.CMD.RegInput1 := FALSE;
   Chain5Long.Drive.ACT.CMD.Brake_Release := FALSE;
   Chain5Long.Drive.ACT.CMD.HwPosOvertravel_Dis := FALSE;
   Chain5Long.Drive.ACT.CMD.HwNegOvertravel_Dis := FALSE;
   Chain5Long.Drive.ACT.CMD.HwOvertravel_MSG_En := FALSE;
   Chain5Long.Drive.ACT.CMD.OneShootMove := FALSE;
   Chain5Long.Drive.ACT.CMD.Move_Type := 3;
   Chain5Long.Drive.ACT.CMD.Target_Pos := 0.0;
   Chain5Long.Drive.ACT.CMD.Speed := 20.0;
   Chain5Long.Drive.ACT.CMD.Acceleration := 300.0;
   Chain5Long.Drive.ACT.CMD.Deceleration := 300.0;
   Chain5Long.Drive.ACT.CMD.Torque_Limit := 30.0;
   Chain5Long.Drive.ACT.CMD.Gear_Ratio := 0.0;
   Chain5Long.Drive.ACT.CMD.Mccp_Length := 2;
   Chain5Long.Drive.ACT.CMD.Mccp_StartSlope := 0.0;
   Chain5Long.Drive.ACT.CMD.Mccp_EndSlope := 0.0;
   Chain5Long.Drive.ACT.CMD.Mapc_Direction := 1;
   Chain5Long.Drive.ACT.CMD.Mapc_SlaveScaling := 1.0;
   Chain5Long.Drive.ACT.CMD.Mapc_MasterScaling := 1.0;
   Chain5Long.Drive.ACT.CMD.Mapc_MasterLockPosition := 0.0;
   Chain5Long.Drive.ACT.CMD.Mapc_CamLockPosition := 0.0;
   Chain5Long.Drive.ACT.CMD.Cam[0].leadingValueStart := 0.0;
   Chain5Long.Drive.ACT.CMD.Cam[1].leadingValueStart := 162.0;
   Chain5Long.Drive.ACT.CMD.Cam[2..39].leadingValueStart := 0.0;
   Chain5Long.Drive.ACT.CMD.Cam[0].leadingValueEnd := 162.0;
   Chain5Long.Drive.ACT.CMD.Cam[1].leadingValueEnd := 360.0;
   Chain5Long.Drive.ACT.CMD.Cam[2..39].leadingValueEnd := 0.0;
   Chain5Long.Drive.ACT.CMD.Cam[0].followingValueStart := 0.0;
   Chain5Long.Drive.ACT.CMD.Cam[1].followingValueStart := 406.399993896484;
   Chain5Long.Drive.ACT.CMD.Cam[2..39].followingValueStart := 0.0;
   Chain5Long.Drive.ACT.CMD.Cam[0..1].followingValueEnd := 406.399993896484;
   Chain5Long.Drive.ACT.CMD.Cam[2..39].followingValueEnd := 0.0;
   Chain5Long.Drive.ACT.CMD.Cam[0..39].geoVeloStart := 0.0;
   Chain5Long.Drive.ACT.CMD.Cam[0..39].geoVeloEnd := 0.0;
   Chain5Long.Drive.ACT.CMD.Cam[0..39].geoAccelStart := 0.0;
   Chain5Long.Drive.ACT.CMD.Cam[0..39].geoAccelEnd := 0.0;
   Chain5Long.Drive.ACT.CMD.Cam[0..39].geoJerkStart := 0.0;
   Chain5Long.Drive.ACT.CMD.Cam[0..39].geoJerkEnd := 0.0;
   Chain5Long.Drive.ACT.CMD.Cam[0..39].inflectionPointParameter := 0.5;
   Chain5Long.Drive.ACT.CMD.Cam[0..39].modVeloTrapezoidParameter := 1.0;
   Chain5Long.Drive.ACT.CMD.Cam[0..39].modSineMaxAccelCaStar := 0.0;
   Chain5Long.Drive.ACT.CMD.Cam[0].camProfileType := 5;
   Chain5Long.Drive.ACT.CMD.Cam[1].camProfileType := 2;
   Chain5Long.Drive.ACT.CMD.Cam[2..39].camProfileType := 0;
   Chain5Long.Drive.ACT.FBK.Ready := TRUE;
   Chain5Long.Drive.ACT.FBK.Calibrated := TRUE;
   Chain5Long.Drive.ACT.FBK.Fault := FALSE;
   Chain5Long.Drive.ACT.FBK.ModuleConnFault := FALSE;
   Chain5Long.Drive.ACT.FBK.In_Position := FALSE;
   Chain5Long.Drive.ACT.FBK.Standstill := TRUE;
   Chain5Long.Drive.ACT.FBK.Enabled := FALSE;
   Chain5Long.Drive.ACT.FBK.BusReadyStatus := FALSE;
   Chain5Long.Drive.ACT.FBK.BrakeReleased := FALSE;
   Chain5Long.Drive.ACT.FBK.HwPosOvertravelDisabled := FALSE;
   Chain5Long.Drive.ACT.FBK.HwNegOvertravelDisabled := FALSE;
   Chain5Long.Drive.ACT.FBK.SafeOffStatus := FALSE;
   Chain5Long.Drive.ACT.FBK.MaxTorqueLimit := FALSE;
   Chain5Long.Drive.ACT.FBK.PosMerge_IP := FALSE;
   Chain5Long.Drive.ACT.FBK.PosMerge_PC := FALSE;
   Chain5Long.Drive.ACT.FBK.Gearing_IP := FALSE;
   Chain5Long.Drive.ACT.FBK.Position := 279.408;
   Chain5Long.Drive.ACT.FBK.Speed := 0.0;
   Chain5Long.Drive.ACT.FBK.Torque := 0.0;
   Chain5Long.Drive.ACT.FBK.RegInput1Pos := 0.0;
   Chain5Long.Drive.ACT.FBK.SeqCamErrorCode := 0;
   Chain5Long.Drive.ACT.FBK.SeqCamTargetPosMAM := 0.0;
   Chain5Long.Drive.ACT.FBK.SeqCamStatus.EndSequence := FALSE;
   Chain5Long.Drive.ACT.FBK.SeqCamStatus.EndSuccess := FALSE;
   Chain5Long.Drive.ACT.FBK.SeqCamStatus.EndError := FALSE;
   Chain5Long.Drive.ACT.FBK.SeqCamStatus.CamHook := FALSE;
   Chain5Long.Drive.ACT.FBK.SeqCamStatus.BothMapc_IP := FALSE;
   Chain5Long.Drive.ACT.FBK.SeqCamStatus.SlaveFwd := FALSE;
   Chain5Long.Drive.ACT.FBK.SeqCamStatus.SlaveBwd := FALSE;
   Chain5Long.Drive.ACT.FBK.SeqCamStatus.SlaveUnwind := FALSE;
   Chain5Long.Drive.ACT.FBK.SeqCamStatus.WaitValidByOpe := FALSE;
   Chain5Long.Drive.ACT.FBK.SeqCamStatus.MapcA_IP := FALSE;
   Chain5Long.Drive.ACT.FBK.SeqCamStatus.MapcB_IP := FALSE;
   Chain5Long.Drive.ACT.FBK.SeqCamStatus.MapcC_IP := FALSE;
   Chain5Long.Drive.ACT.FBK.SeqCamStatus.CamOnce_PC := FALSE;
   Chain5Long.Drive.ACT.FBK.SeqCamStatus.MaxDevError := FALSE;
   Chain5Long.Drive.ACT.FBK.SeqCamStatus.PositionCamLockStatus := FALSE;
   Chain5Long.Drive.ACT.FBK.SeqCamStatus.WaitRestart := FALSE;
   Chain5Long.Drive.ACT.FBK.SeqCamStatus.Bit17 := FALSE;
   Chain5Long.Drive.ACT.FBK.SeqCamStatus.Bit18 := FALSE;
   Chain5Long.Drive.ACT.FBK.SeqCamStatus.Bit19 := FALSE;
   Chain5Long.Drive.ACT.FBK.SeqCamStatus.Bit20 := FALSE;
   Chain5Long.Drive.ACT.FBK.SeqCamStatus.Bit21 := FALSE;
   Chain5Long.Drive.ACT.FBK.SeqCamStatus.Bit22 := FALSE;
   Chain5Long.Drive.ACT.FBK.SeqCamStatus.Bit23 := FALSE;
   Chain5Long.Drive.ACT.FBK.SeqCamStatus.Bit24 := FALSE;
   Chain5Long.Drive.ACT.FBK.SeqCamStatus.Bit25 := FALSE;
   Chain5Long.Drive.ACT.FBK.SeqCamStatus.Bit26 := FALSE;
   Chain5Long.Drive.ACT.FBK.SeqCamStatus.Bit27 := FALSE;
   Chain5Long.Drive.ACT.FBK.SeqCamStatus.Bit28 := FALSE;
   Chain5Long.Drive.ACT.FBK.SeqCamStatus.Bit29 := FALSE;
   Chain5Long.Drive.ACT.FBK.SeqCamStatus.Bit30 := FALSE;
   Chain5Long.Drive.ACT.FBK.SeqCamStatus.Bit31 := FALSE;
   Chain5Long.Drive.ACT.FBK.SeqCamStatus.Bit32 := FALSE;
   Chain5Long.Drive.PLS.FinePosOk.LowLimit := 405.4;
   Chain5Long.Drive.PLS.FinePosOk.HighLimit := 1.0;
   Chain5Long.Drive.PLS.FinePosOk.Ok := FALSE;
   Chain5Long.Drive.PLS.KeepPosOk.LowLimit := 404.4;
   Chain5Long.Drive.PLS.KeepPosOk.HighLimit := 2.0;
   Chain5Long.Drive.PLS.KeepPosOk.Ok := FALSE;
   Chain5Long.Drive.PLS.Up.LowLimit := 0.0;
   Chain5Long.Drive.PLS.Up.HighLimit := 0.0;
   Chain5Long.Drive.PLS.Up.Ok := FALSE;
   Chain5Long.Drive.PLS.Intermediate.LowLimit := 0.0;
   Chain5Long.Drive.PLS.Intermediate.HighLimit := 0.0;
   Chain5Long.Drive.PLS.Intermediate.Ok := FALSE;
   Chain5Long.Drive.PLS.Down.LowLimit := 0.0;
   Chain5Long.Drive.PLS.Down.HighLimit := 0.0;
   Chain5Long.Drive.PLS.Down.Ok := FALSE;
   Chain5Long.Drive.PLS.Forward.LowLimit := 0.0;
   Chain5Long.Drive.PLS.Forward.HighLimit := 0.0;
   Chain5Long.Drive.PLS.Forward.Ok := FALSE;
   Chain5Long.Drive.PLS.Backward.LowLimit := 0.0;
   Chain5Long.Drive.PLS.Backward.HighLimit := 0.0;
   Chain5Long.Drive.PLS.Backward.Ok := FALSE;
   Chain5Long.Drive.PLS.Open.LowLimit := 0.0;
   Chain5Long.Drive.PLS.Open.HighLimit := 0.0;
   Chain5Long.Drive.PLS.Open.Ok := FALSE;
   Chain5Long.Drive.PLS.Close.LowLimit := 0.0;
   Chain5Long.Drive.PLS.Close.HighLimit := 0.0;
   Chain5Long.Drive.PLS.Close.Ok := FALSE;
   Chain5Long.Drive.PLS.PreOpen.LowLimit := 0.0;
   Chain5Long.Drive.PLS.PreOpen.HighLimit := 0.0;
   Chain5Long.Drive.PLS.PreOpen.Ok := FALSE;
   Chain5Long.Drive.PLS.Maintenance.LowLimit := 0.0;
   Chain5Long.Drive.PLS.Maintenance.HighLimit := 0.0;
   Chain5Long.Drive.PLS.Maintenance.Ok := FALSE;
   Chain5Long.Drive.PLS.OperatorSide.LowLimit := 0.0;
   Chain5Long.Drive.PLS.OperatorSide.HighLimit := 0.0;
   Chain5Long.Drive.PLS.OperatorSide.Ok := FALSE;
   Chain5Long.Drive.PLS.NotOperatorSide.LowLimit := 0.0;
   Chain5Long.Drive.PLS.NotOperatorSide.HighLimit := 0.0;
   Chain5Long.Drive.PLS.NotOperatorSide.Ok := FALSE;
   Chain5Long.Drive.PLS.OnMould.LowLimit := 0.0;
   Chain5Long.Drive.PLS.OnMould.HighLimit := 0.0;
   Chain5Long.Drive.PLS.OnMould.Ok := FALSE;
   Chain5Long.Drive.PLS.OffMould.LowLimit := 0.0;
   Chain5Long.Drive.PLS.OffMould.HighLimit := 0.0;
   Chain5Long.Drive.PLS.OffMould.Ok := FALSE;
   Chain5Long.Drive.PLS.Pos0.LowLimit := 0.0;
   Chain5Long.Drive.PLS.Pos0.HighLimit := 0.0;
   Chain5Long.Drive.PLS.Pos0.Ok := FALSE;
   Chain5Long.Drive.PLS.Pos1.LowLimit := 0.0;
   Chain5Long.Drive.PLS.Pos1.HighLimit := 0.0;
   Chain5Long.Drive.PLS.Pos1.Ok := FALSE;
   Chain5Long.Drive.PLS.Pos2.LowLimit := 0.0;
   Chain5Long.Drive.PLS.Pos2.HighLimit := 0.0;
   Chain5Long.Drive.PLS.Pos2.Ok := FALSE;
   Chain5Long.Drive.PLS.Pos3.LowLimit := 0.0;
   Chain5Long.Drive.PLS.Pos3.HighLimit := 0.0;
   Chain5Long.Drive.PLS.Pos3.Ok := FALSE;
   Chain5Long.Drive.PLS.Pos4.LowLimit := 0.0;
   Chain5Long.Drive.PLS.Pos4.HighLimit := 0.0;
   Chain5Long.Drive.PLS.Pos4.Ok := FALSE;
   Chain5Long.Drive.PLS.Pos5.LowLimit := 0.0;
   Chain5Long.Drive.PLS.Pos5.HighLimit := 0.0;
   Chain5Long.Drive.PLS.Pos5.Ok := FALSE;
   Chain5Long.Drive.TON_EnableDrive.PT := T#500MS;
   Chain5Long.Drive.TON_EnableDrive.IN := FALSE;
   Chain5Long.Drive.TON_HwOvertravel_Dis.PT := T#0MS;
   Chain5Long.Drive.TON_HwOvertravel_Dis.IN := FALSE;
   Chain5Long.Drive.TON_HwOvertravel_En.PT := T#0MS;
   Chain5Long.Drive.TON_HwOvertravel_En.IN := FALSE;
   Chain5Long.Drive.TON_TimeoutMovement.PT := T#0MS;
   Chain5Long.Drive.TON_TimeoutMovement.IN := FALSE;
   Chain6Long.AlmOk := TRUE;
   Chain6Long.StationWorked := TRUE;
   Chain6Long.CheckObstruction := TRUE;
   Chain6Long.OutChainObstruction := TRUE;
   Chain6Long.StrobeWork := FALSE;
   Chain6Long.StrobeShift := FALSE;
   Chain6Long.ManualMovement := FALSE;
   Chain6Long.OkToStop := TRUE;
   Chain6Long.PosOk := FALSE;
   Chain6Long.Ons_PosOk := FALSE;
   Chain6Long.EnaMove := TRUE;
   Chain6Long.StationEna := FALSE;
   Chain6Long.ModeLong := TRUE;
   Chain6Long.ModeCross := FALSE;
   Chain6Long.ModeCont := FALSE;
   Chain6Long.Cfg_Mould_ChainSteps := 1;
   Chain6Long.Cfg_Mould_EndPos := 1;
   Chain6Long.Shift_Lenght := 2;
   Chain6Long.PosMasterAdvanceStep := 0.0;
   Chain6Long.Input.EndChaMouPre := FALSE;
   Chain6Long.Input.PshHig := FALSE;
   Chain6Long.Input.PshLow := FALSE;
   Chain6Long.Output.PshHig := FALSE;
   Chain6Long.Output.PshLow := FALSE;
   Chain6Long.Man.EnaPbt := FALSE;
   Chain6Long.Man.RstCmd := TRUE;
   Chain6Long.Man.ScreenNumber := 300_060_301;
   Chain6Long.Man.WithinScreenRange := 0;
   Chain6Long.Drive.AlmOk := FALSE;
   Chain6Long.Drive.AlmEmerg := FALSE;
   Chain6Long.Drive.AlmNode := FALSE;
   Chain6Long.Drive.InitPosDrive := FALSE;
   Chain6Long.Drive.InitPosDrivePLS := FALSE;
   Chain6Long.Drive.GearingON := FALSE;
   Chain6Long.Drive.CamHook := FALSE;
   Chain6Long.Drive.CamStoppingPhase := FALSE;
   Chain6Long.Drive.RepositioningRequest := FALSE;
   Chain6Long.Drive.CamRequestResult := FALSE;
   Chain6Long.Drive.CamRequestError := FALSE;
   Chain6Long.Drive.CamRequestOk := TRUE;
   Chain6Long.Drive.CalibDisAxisReq := FALSE;
   Chain6Long.Drive.CalibReq := FALSE;
   Chain6Long.Drive.CalibProcess := FALSE;
   Chain6Long.Drive.HwOvertravelDisReq := FALSE;
   Chain6Long.Drive.HwOvertravelEnReq := FALSE;
   Chain6Long.Drive.AuxCamRequest := FALSE;
   Chain6Long.Drive.TorquePeakEna := TRUE;
   Chain6Long.Drive.Cmd_Repos := FALSE;
   Chain6Long.Drive.Ons_CamRequest := FALSE;
   Chain6Long.Drive.AuxCmdPosition := 0;
   Chain6Long.Drive.Unwind := 406.4;
   Chain6Long.Drive.MaxDev := 150.0;
   Chain6Long.Drive.ReposSpeed := 10.0;
   Chain6Long.Drive.CalcSlaveDifferenceABS := 0.0;
   Chain6Long.Drive.CalcModPosition := 0.0;
   Chain6Long.Drive.CalcSlaveDifference := 0.0;
   Chain6Long.Drive.CalcMinDeltaPos := 0.0;
   Chain6Long.Drive.CalcMaxDeltaPos := 0.0;
   Chain6Long.Drive.CalcHalfPosUnwind := 0.0;
   Chain6Long.Drive.Man.Cmd_PosJog := FALSE;
   Chain6Long.Drive.Man.Cmd_NegJog := FALSE;
   Chain6Long.Drive.Man.Cmd_Step := FALSE;
   Chain6Long.Drive.Man.Cmd_Forward := FALSE;
   Chain6Long.Drive.Man.Cmd_Backward := FALSE;
   Chain6Long.Drive.Man.Cmd_Up := FALSE;
   Chain6Long.Drive.Man.Cmd_Down := FALSE;
   Chain6Long.Drive.Man.Cmd_Intermediate := FALSE;
   Chain6Long.Drive.Man.Cmd_Open := FALSE;
   Chain6Long.Drive.Man.Cmd_Close := FALSE;
   Chain6Long.Drive.Man.Cmd_PreOpen := FALSE;
   Chain6Long.Drive.Man.Cmd_Maintenance := FALSE;
   Chain6Long.Drive.Man.Cmd_OperatorSide := FALSE;
   Chain6Long.Drive.Man.Cmd_NotOperatorSide := FALSE;
   Chain6Long.Drive.Man.Cmd_OnMould := FALSE;
   Chain6Long.Drive.Man.Cmd_OffMould := FALSE;
   Chain6Long.Drive.Man.Cmd_Pos0 := FALSE;
   Chain6Long.Drive.Man.Cmd_Pos1 := FALSE;
   Chain6Long.Drive.Man.Cmd_Pos2 := FALSE;
   Chain6Long.Drive.Man.Cmd_Pos3 := FALSE;
   Chain6Long.Drive.Man.Cmd_Pos4 := FALSE;
   Chain6Long.Drive.Man.Cmd_Pos5 := FALSE;
   Chain6Long.Drive.Man.Ons_Step := FALSE;
   Chain6Long.Drive.Man.PhaseJogCmd := FALSE;
   Chain6Long.Drive.Man.CmdStartStep := FALSE;
   Chain6Long.Drive.Man.CmdEndStep := FALSE;
   Chain6Long.Drive.Man.StepCond := FALSE;
   Chain6Long.Drive.Man.TON_DelayHomeCmd.PT := T#3S;
   Chain6Long.Drive.Man.TON_DelayHomeCmd.IN := FALSE;
   Chain6Long.Drive.Auto.Cmd_Step := FALSE;
   Chain6Long.Drive.Auto.Cmd_StartStep := FALSE;
   Chain6Long.Drive.Auto.Cmd_EndStep := FALSE;
   Chain6Long.Drive.Auto.Cmd_Forward := FALSE;
   Chain6Long.Drive.Auto.Cmd_Backward := FALSE;
   Chain6Long.Drive.Auto.Cmd_Up := FALSE;
   Chain6Long.Drive.Auto.Cmd_Down := FALSE;
   Chain6Long.Drive.Auto.Cmd_Intermediate := FALSE;
   Chain6Long.Drive.Auto.Cmd_Open := FALSE;
   Chain6Long.Drive.Auto.Cmd_Close := FALSE;
   Chain6Long.Drive.Auto.Cmd_PreOpen := FALSE;
   Chain6Long.Drive.Auto.Cmd_Maintenance := FALSE;
   Chain6Long.Drive.Auto.Cmd_OperatorSide := FALSE;
   Chain6Long.Drive.Auto.Cmd_NotOperatorSide := FALSE;
   Chain6Long.Drive.Auto.Cmd_OnMould := FALSE;
   Chain6Long.Drive.Auto.Cmd_OffMould := FALSE;
   Chain6Long.Drive.Auto.Cmd_Pos0 := FALSE;
   Chain6Long.Drive.Auto.Cmd_Pos1 := FALSE;
   Chain6Long.Drive.Auto.Cmd_Pos2 := FALSE;
   Chain6Long.Drive.Auto.Cmd_Pos3 := FALSE;
   Chain6Long.Drive.Auto.Cmd_Pos4 := FALSE;
   Chain6Long.Drive.Auto.Cmd_Pos5 := FALSE;
   Chain6Long.Drive.Auto.Cmd_Gear := FALSE;
   Chain6Long.Drive.ACT.CMD.Enable := FALSE;
   Chain6Long.Drive.ACT.CMD.Pos_Mode := FALSE;
   Chain6Long.Drive.ACT.CMD.MergeDisabled := FALSE;
   Chain6Long.Drive.ACT.CMD.SCurve := FALSE;
   Chain6Long.Drive.ACT.CMD.Cam_Mode := TRUE;
   Chain6Long.Drive.ACT.CMD.Cam_Request := FALSE;
   Chain6Long.Drive.ACT.CMD.Cam_PhaseStop := FALSE;
   Chain6Long.Drive.ACT.CMD.Gear_Mode := FALSE;
   Chain6Long.Drive.ACT.CMD.Repos_Req := FALSE;
   Chain6Long.Drive.ACT.CMD.Jog_Pos := FALSE;
   Chain6Long.Drive.ACT.CMD.Jog_Neg := FALSE;
   Chain6Long.Drive.ACT.CMD.Stop := FALSE;
   Chain6Long.Drive.ACT.CMD.Calibration_Req := FALSE;
   Chain6Long.Drive.ACT.CMD.Reset := FALSE;
   Chain6Long.Drive.ACT.CMD.RegInput1 := FALSE;
   Chain6Long.Drive.ACT.CMD.Brake_Release := FALSE;
   Chain6Long.Drive.ACT.CMD.HwPosOvertravel_Dis := FALSE;
   Chain6Long.Drive.ACT.CMD.HwNegOvertravel_Dis := FALSE;
   Chain6Long.Drive.ACT.CMD.HwOvertravel_MSG_En := FALSE;
   Chain6Long.Drive.ACT.CMD.OneShootMove := FALSE;
   Chain6Long.Drive.ACT.CMD.Move_Type := 3;
   Chain6Long.Drive.ACT.CMD.Target_Pos := 0.0;
   Chain6Long.Drive.ACT.CMD.Speed := 5.0;
   Chain6Long.Drive.ACT.CMD.Acceleration := 300.0;
   Chain6Long.Drive.ACT.CMD.Deceleration := 300.0;
   Chain6Long.Drive.ACT.CMD.Torque_Limit := 30.0;
   Chain6Long.Drive.ACT.CMD.Gear_Ratio := 0.0;
   Chain6Long.Drive.ACT.CMD.Mccp_Length := 2;
   Chain6Long.Drive.ACT.CMD.Mccp_StartSlope := 0.0;
   Chain6Long.Drive.ACT.CMD.Mccp_EndSlope := 0.0;
   Chain6Long.Drive.ACT.CMD.Mapc_Direction := 1;
   Chain6Long.Drive.ACT.CMD.Mapc_SlaveScaling := 1.0;
   Chain6Long.Drive.ACT.CMD.Mapc_MasterScaling := 1.0;
   Chain6Long.Drive.ACT.CMD.Mapc_MasterLockPosition := 0.0;
   Chain6Long.Drive.ACT.CMD.Mapc_CamLockPosition := 0.0;
   Chain6Long.Drive.ACT.CMD.Cam[0].leadingValueStart := 0.0;
   Chain6Long.Drive.ACT.CMD.Cam[1].leadingValueStart := 162.0;
   Chain6Long.Drive.ACT.CMD.Cam[2..39].leadingValueStart := 0.0;
   Chain6Long.Drive.ACT.CMD.Cam[0].leadingValueEnd := 162.0;
   Chain6Long.Drive.ACT.CMD.Cam[1].leadingValueEnd := 360.0;
   Chain6Long.Drive.ACT.CMD.Cam[2..39].leadingValueEnd := 0.0;
   Chain6Long.Drive.ACT.CMD.Cam[0].followingValueStart := 0.0;
   Chain6Long.Drive.ACT.CMD.Cam[1].followingValueStart := 406.399993896484;
   Chain6Long.Drive.ACT.CMD.Cam[2..39].followingValueStart := 0.0;
   Chain6Long.Drive.ACT.CMD.Cam[0..1].followingValueEnd := 406.399993896484;
   Chain6Long.Drive.ACT.CMD.Cam[2..39].followingValueEnd := 0.0;
   Chain6Long.Drive.ACT.CMD.Cam[0..39].geoVeloStart := 0.0;
   Chain6Long.Drive.ACT.CMD.Cam[0..39].geoVeloEnd := 0.0;
   Chain6Long.Drive.ACT.CMD.Cam[0..39].geoAccelStart := 0.0;
   Chain6Long.Drive.ACT.CMD.Cam[0..39].geoAccelEnd := 0.0;
   Chain6Long.Drive.ACT.CMD.Cam[0..39].geoJerkStart := 0.0;
   Chain6Long.Drive.ACT.CMD.Cam[0..39].geoJerkEnd := 0.0;
   Chain6Long.Drive.ACT.CMD.Cam[0..39].inflectionPointParameter := 0.5;
   Chain6Long.Drive.ACT.CMD.Cam[0..39].modVeloTrapezoidParameter := 1.0;
   Chain6Long.Drive.ACT.CMD.Cam[0..39].modSineMaxAccelCaStar := 0.0;
   Chain6Long.Drive.ACT.CMD.Cam[0].camProfileType := 5;
   Chain6Long.Drive.ACT.CMD.Cam[1].camProfileType := 2;
   Chain6Long.Drive.ACT.CMD.Cam[2..39].camProfileType := 0;
   Chain6Long.Drive.ACT.FBK.Ready := TRUE;
   Chain6Long.Drive.ACT.FBK.Calibrated := TRUE;
   Chain6Long.Drive.ACT.FBK.Fault := FALSE;
   Chain6Long.Drive.ACT.FBK.ModuleConnFault := FALSE;
   Chain6Long.Drive.ACT.FBK.In_Position := FALSE;
   Chain6Long.Drive.ACT.FBK.Standstill := TRUE;
   Chain6Long.Drive.ACT.FBK.Enabled := FALSE;
   Chain6Long.Drive.ACT.FBK.BusReadyStatus := FALSE;
   Chain6Long.Drive.ACT.FBK.BrakeReleased := FALSE;
   Chain6Long.Drive.ACT.FBK.HwPosOvertravelDisabled := FALSE;
   Chain6Long.Drive.ACT.FBK.HwNegOvertravelDisabled := FALSE;
   Chain6Long.Drive.ACT.FBK.SafeOffStatus := FALSE;
   Chain6Long.Drive.ACT.FBK.MaxTorqueLimit := FALSE;
   Chain6Long.Drive.ACT.FBK.PosMerge_IP := FALSE;
   Chain6Long.Drive.ACT.FBK.PosMerge_PC := FALSE;
   Chain6Long.Drive.ACT.FBK.Gearing_IP := FALSE;
   Chain6Long.Drive.ACT.FBK.Position := 279.461;
   Chain6Long.Drive.ACT.FBK.Speed := -0.006435854;
   Chain6Long.Drive.ACT.FBK.Torque := 0.02441406;
   Chain6Long.Drive.ACT.FBK.RegInput1Pos := 0.0;
   Chain6Long.Drive.ACT.FBK.SeqCamErrorCode := 0;
   Chain6Long.Drive.ACT.FBK.SeqCamTargetPosMAM := 0.0;
   Chain6Long.Drive.ACT.FBK.SeqCamStatus.EndSequence := FALSE;
   Chain6Long.Drive.ACT.FBK.SeqCamStatus.EndSuccess := FALSE;
   Chain6Long.Drive.ACT.FBK.SeqCamStatus.EndError := FALSE;
   Chain6Long.Drive.ACT.FBK.SeqCamStatus.CamHook := FALSE;
   Chain6Long.Drive.ACT.FBK.SeqCamStatus.BothMapc_IP := FALSE;
   Chain6Long.Drive.ACT.FBK.SeqCamStatus.SlaveFwd := FALSE;
   Chain6Long.Drive.ACT.FBK.SeqCamStatus.SlaveBwd := FALSE;
   Chain6Long.Drive.ACT.FBK.SeqCamStatus.SlaveUnwind := FALSE;
   Chain6Long.Drive.ACT.FBK.SeqCamStatus.WaitValidByOpe := FALSE;
   Chain6Long.Drive.ACT.FBK.SeqCamStatus.MapcA_IP := FALSE;
   Chain6Long.Drive.ACT.FBK.SeqCamStatus.MapcB_IP := FALSE;
   Chain6Long.Drive.ACT.FBK.SeqCamStatus.MapcC_IP := FALSE;
   Chain6Long.Drive.ACT.FBK.SeqCamStatus.CamOnce_PC := FALSE;
   Chain6Long.Drive.ACT.FBK.SeqCamStatus.MaxDevError := FALSE;
   Chain6Long.Drive.ACT.FBK.SeqCamStatus.PositionCamLockStatus := FALSE;
   Chain6Long.Drive.ACT.FBK.SeqCamStatus.WaitRestart := FALSE;
   Chain6Long.Drive.ACT.FBK.SeqCamStatus.Bit17 := FALSE;
   Chain6Long.Drive.ACT.FBK.SeqCamStatus.Bit18 := FALSE;
   Chain6Long.Drive.ACT.FBK.SeqCamStatus.Bit19 := FALSE;
   Chain6Long.Drive.ACT.FBK.SeqCamStatus.Bit20 := FALSE;
   Chain6Long.Drive.ACT.FBK.SeqCamStatus.Bit21 := FALSE;
   Chain6Long.Drive.ACT.FBK.SeqCamStatus.Bit22 := FALSE;
   Chain6Long.Drive.ACT.FBK.SeqCamStatus.Bit23 := FALSE;
   Chain6Long.Drive.ACT.FBK.SeqCamStatus.Bit24 := FALSE;
   Chain6Long.Drive.ACT.FBK.SeqCamStatus.Bit25 := FALSE;
   Chain6Long.Drive.ACT.FBK.SeqCamStatus.Bit26 := FALSE;
   Chain6Long.Drive.ACT.FBK.SeqCamStatus.Bit27 := FALSE;
   Chain6Long.Drive.ACT.FBK.SeqCamStatus.Bit28 := FALSE;
   Chain6Long.Drive.ACT.FBK.SeqCamStatus.Bit29 := FALSE;
   Chain6Long.Drive.ACT.FBK.SeqCamStatus.Bit30 := FALSE;
   Chain6Long.Drive.ACT.FBK.SeqCamStatus.Bit31 := FALSE;
   Chain6Long.Drive.ACT.FBK.SeqCamStatus.Bit32 := FALSE;
   Chain6Long.Drive.PLS.FinePosOk.LowLimit := 405.4;
   Chain6Long.Drive.PLS.FinePosOk.HighLimit := 1.0;
   Chain6Long.Drive.PLS.FinePosOk.Ok := FALSE;
   Chain6Long.Drive.PLS.KeepPosOk.LowLimit := 404.4;
   Chain6Long.Drive.PLS.KeepPosOk.HighLimit := 2.0;
   Chain6Long.Drive.PLS.KeepPosOk.Ok := FALSE;
   Chain6Long.Drive.PLS.Up.LowLimit := 0.0;
   Chain6Long.Drive.PLS.Up.HighLimit := 0.0;
   Chain6Long.Drive.PLS.Up.Ok := FALSE;
   Chain6Long.Drive.PLS.Intermediate.LowLimit := 0.0;
   Chain6Long.Drive.PLS.Intermediate.HighLimit := 0.0;
   Chain6Long.Drive.PLS.Intermediate.Ok := FALSE;
   Chain6Long.Drive.PLS.Down.LowLimit := 0.0;
   Chain6Long.Drive.PLS.Down.HighLimit := 0.0;
   Chain6Long.Drive.PLS.Down.Ok := FALSE;
   Chain6Long.Drive.PLS.Forward.LowLimit := 0.0;
   Chain6Long.Drive.PLS.Forward.HighLimit := 0.0;
   Chain6Long.Drive.PLS.Forward.Ok := FALSE;
   Chain6Long.Drive.PLS.Backward.LowLimit := 0.0;
   Chain6Long.Drive.PLS.Backward.HighLimit := 0.0;
   Chain6Long.Drive.PLS.Backward.Ok := FALSE;
   Chain6Long.Drive.PLS.Open.LowLimit := 0.0;
   Chain6Long.Drive.PLS.Open.HighLimit := 0.0;
   Chain6Long.Drive.PLS.Open.Ok := FALSE;
   Chain6Long.Drive.PLS.Close.LowLimit := 0.0;
   Chain6Long.Drive.PLS.Close.HighLimit := 0.0;
   Chain6Long.Drive.PLS.Close.Ok := FALSE;
   Chain6Long.Drive.PLS.PreOpen.LowLimit := 0.0;
   Chain6Long.Drive.PLS.PreOpen.HighLimit := 0.0;
   Chain6Long.Drive.PLS.PreOpen.Ok := FALSE;
   Chain6Long.Drive.PLS.Maintenance.LowLimit := 0.0;
   Chain6Long.Drive.PLS.Maintenance.HighLimit := 0.0;
   Chain6Long.Drive.PLS.Maintenance.Ok := FALSE;
   Chain6Long.Drive.PLS.OperatorSide.LowLimit := 0.0;
   Chain6Long.Drive.PLS.OperatorSide.HighLimit := 0.0;
   Chain6Long.Drive.PLS.OperatorSide.Ok := FALSE;
   Chain6Long.Drive.PLS.NotOperatorSide.LowLimit := 0.0;
   Chain6Long.Drive.PLS.NotOperatorSide.HighLimit := 0.0;
   Chain6Long.Drive.PLS.NotOperatorSide.Ok := FALSE;
   Chain6Long.Drive.PLS.OnMould.LowLimit := 0.0;
   Chain6Long.Drive.PLS.OnMould.HighLimit := 0.0;
   Chain6Long.Drive.PLS.OnMould.Ok := FALSE;
   Chain6Long.Drive.PLS.OffMould.LowLimit := 0.0;
   Chain6Long.Drive.PLS.OffMould.HighLimit := 0.0;
   Chain6Long.Drive.PLS.OffMould.Ok := FALSE;
   Chain6Long.Drive.PLS.Pos0.LowLimit := 0.0;
   Chain6Long.Drive.PLS.Pos0.HighLimit := 0.0;
   Chain6Long.Drive.PLS.Pos0.Ok := FALSE;
   Chain6Long.Drive.PLS.Pos1.LowLimit := 0.0;
   Chain6Long.Drive.PLS.Pos1.HighLimit := 0.0;
   Chain6Long.Drive.PLS.Pos1.Ok := FALSE;
   Chain6Long.Drive.PLS.Pos2.LowLimit := 0.0;
   Chain6Long.Drive.PLS.Pos2.HighLimit := 0.0;
   Chain6Long.Drive.PLS.Pos2.Ok := FALSE;
   Chain6Long.Drive.PLS.Pos3.LowLimit := 0.0;
   Chain6Long.Drive.PLS.Pos3.HighLimit := 0.0;
   Chain6Long.Drive.PLS.Pos3.Ok := FALSE;
   Chain6Long.Drive.PLS.Pos4.LowLimit := 0.0;
   Chain6Long.Drive.PLS.Pos4.HighLimit := 0.0;
   Chain6Long.Drive.PLS.Pos4.Ok := FALSE;
   Chain6Long.Drive.PLS.Pos5.LowLimit := 0.0;
   Chain6Long.Drive.PLS.Pos5.HighLimit := 0.0;
   Chain6Long.Drive.PLS.Pos5.Ok := FALSE;
   Chain6Long.Drive.TON_EnableDrive.PT := T#500MS;
   Chain6Long.Drive.TON_EnableDrive.IN := FALSE;
   Chain6Long.Drive.TON_HwOvertravel_Dis.PT := T#0MS;
   Chain6Long.Drive.TON_HwOvertravel_Dis.IN := FALSE;
   Chain6Long.Drive.TON_HwOvertravel_En.PT := T#0MS;
   Chain6Long.Drive.TON_HwOvertravel_En.IN := FALSE;
   Chain6Long.Drive.TON_TimeoutMovement.PT := T#0MS;
   Chain6Long.Drive.TON_TimeoutMovement.IN := FALSE;
   Chain7Long.AlmOk := TRUE;
   Chain7Long.StationWorked := TRUE;
   Chain7Long.CheckObstruction := TRUE;
   Chain7Long.OutChainObstruction := TRUE;
   Chain7Long.StrobeWork := FALSE;
   Chain7Long.StrobeShift := FALSE;
   Chain7Long.ManualMovement := FALSE;
   Chain7Long.OkToStop := TRUE;
   Chain7Long.PosOk := FALSE;
   Chain7Long.Ons_PosOk := FALSE;
   Chain7Long.EnaMove := TRUE;
   Chain7Long.StationEna := FALSE;
   Chain7Long.ModeLong := TRUE;
   Chain7Long.ModeCross := FALSE;
   Chain7Long.ModeCont := FALSE;
   Chain7Long.Cfg_Mould_ChainSteps := 1;
   Chain7Long.Cfg_Mould_EndPos := 31;
   Chain7Long.Shift_Lenght := 32;
   Chain7Long.PosMasterAdvanceStep := 0.0;
   Chain7Long.Input.EndChaMouPre := FALSE;
   Chain7Long.Input.PshHig := FALSE;
   Chain7Long.Input.PshLow := FALSE;
   Chain7Long.Output.PshHig := FALSE;
   Chain7Long.Output.PshLow := FALSE;
   Chain7Long.Man.EnaPbt := FALSE;
   Chain7Long.Man.RstCmd := TRUE;
   Chain7Long.Man.ScreenNumber := 300_070_301;
   Chain7Long.Man.WithinScreenRange := 0;
   Chain7Long.Drive.AlmOk := FALSE;
   Chain7Long.Drive.AlmEmerg := FALSE;
   Chain7Long.Drive.AlmNode := FALSE;
   Chain7Long.Drive.InitPosDrive := FALSE;
   Chain7Long.Drive.InitPosDrivePLS := FALSE;
   Chain7Long.Drive.GearingON := FALSE;
   Chain7Long.Drive.CamHook := FALSE;
   Chain7Long.Drive.CamStoppingPhase := FALSE;
   Chain7Long.Drive.RepositioningRequest := FALSE;
   Chain7Long.Drive.CamRequestResult := FALSE;
   Chain7Long.Drive.CamRequestError := FALSE;
   Chain7Long.Drive.CamRequestOk := TRUE;
   Chain7Long.Drive.CalibDisAxisReq := FALSE;
   Chain7Long.Drive.CalibReq := FALSE;
   Chain7Long.Drive.CalibProcess := FALSE;
   Chain7Long.Drive.HwOvertravelDisReq := FALSE;
   Chain7Long.Drive.HwOvertravelEnReq := FALSE;
   Chain7Long.Drive.AuxCamRequest := FALSE;
   Chain7Long.Drive.TorquePeakEna := TRUE;
   Chain7Long.Drive.Cmd_Repos := FALSE;
   Chain7Long.Drive.Ons_CamRequest := FALSE;
   Chain7Long.Drive.AuxCmdPosition := 0;
   Chain7Long.Drive.Unwind := 406.4;
   Chain7Long.Drive.MaxDev := 150.0;
   Chain7Long.Drive.ReposSpeed := 10.0;
   Chain7Long.Drive.CalcSlaveDifferenceABS := 0.0;
   Chain7Long.Drive.CalcModPosition := 0.0;
   Chain7Long.Drive.CalcSlaveDifference := 0.0;
   Chain7Long.Drive.CalcMinDeltaPos := 0.0;
   Chain7Long.Drive.CalcMaxDeltaPos := 0.0;
   Chain7Long.Drive.CalcHalfPosUnwind := 0.0;
   Chain7Long.Drive.Man.Cmd_PosJog := FALSE;
   Chain7Long.Drive.Man.Cmd_NegJog := FALSE;
   Chain7Long.Drive.Man.Cmd_Step := FALSE;
   Chain7Long.Drive.Man.Cmd_Forward := FALSE;
   Chain7Long.Drive.Man.Cmd_Backward := FALSE;
   Chain7Long.Drive.Man.Cmd_Up := FALSE;
   Chain7Long.Drive.Man.Cmd_Down := FALSE;
   Chain7Long.Drive.Man.Cmd_Intermediate := FALSE;
   Chain7Long.Drive.Man.Cmd_Open := FALSE;
   Chain7Long.Drive.Man.Cmd_Close := FALSE;
   Chain7Long.Drive.Man.Cmd_PreOpen := FALSE;
   Chain7Long.Drive.Man.Cmd_Maintenance := FALSE;
   Chain7Long.Drive.Man.Cmd_OperatorSide := FALSE;
   Chain7Long.Drive.Man.Cmd_NotOperatorSide := FALSE;
   Chain7Long.Drive.Man.Cmd_OnMould := FALSE;
   Chain7Long.Drive.Man.Cmd_OffMould := FALSE;
   Chain7Long.Drive.Man.Cmd_Pos0 := FALSE;
   Chain7Long.Drive.Man.Cmd_Pos1 := FALSE;
   Chain7Long.Drive.Man.Cmd_Pos2 := FALSE;
   Chain7Long.Drive.Man.Cmd_Pos3 := FALSE;
   Chain7Long.Drive.Man.Cmd_Pos4 := FALSE;
   Chain7Long.Drive.Man.Cmd_Pos5 := FALSE;
   Chain7Long.Drive.Man.Ons_Step := FALSE;
   Chain7Long.Drive.Man.PhaseJogCmd := FALSE;
   Chain7Long.Drive.Man.CmdStartStep := FALSE;
   Chain7Long.Drive.Man.CmdEndStep := FALSE;
   Chain7Long.Drive.Man.StepCond := FALSE;
   Chain7Long.Drive.Man.TON_DelayHomeCmd.PT := T#3S;
   Chain7Long.Drive.Man.TON_DelayHomeCmd.IN := FALSE;
   Chain7Long.Drive.Auto.Cmd_Step := FALSE;
   Chain7Long.Drive.Auto.Cmd_StartStep := FALSE;
   Chain7Long.Drive.Auto.Cmd_EndStep := FALSE;
   Chain7Long.Drive.Auto.Cmd_Forward := FALSE;
   Chain7Long.Drive.Auto.Cmd_Backward := FALSE;
   Chain7Long.Drive.Auto.Cmd_Up := FALSE;
   Chain7Long.Drive.Auto.Cmd_Down := FALSE;
   Chain7Long.Drive.Auto.Cmd_Intermediate := FALSE;
   Chain7Long.Drive.Auto.Cmd_Open := FALSE;
   Chain7Long.Drive.Auto.Cmd_Close := FALSE;
   Chain7Long.Drive.Auto.Cmd_PreOpen := FALSE;
   Chain7Long.Drive.Auto.Cmd_Maintenance := FALSE;
   Chain7Long.Drive.Auto.Cmd_OperatorSide := FALSE;
   Chain7Long.Drive.Auto.Cmd_NotOperatorSide := FALSE;
   Chain7Long.Drive.Auto.Cmd_OnMould := FALSE;
   Chain7Long.Drive.Auto.Cmd_OffMould := FALSE;
   Chain7Long.Drive.Auto.Cmd_Pos0 := FALSE;
   Chain7Long.Drive.Auto.Cmd_Pos1 := FALSE;
   Chain7Long.Drive.Auto.Cmd_Pos2 := FALSE;
   Chain7Long.Drive.Auto.Cmd_Pos3 := FALSE;
   Chain7Long.Drive.Auto.Cmd_Pos4 := FALSE;
   Chain7Long.Drive.Auto.Cmd_Pos5 := FALSE;
   Chain7Long.Drive.Auto.Cmd_Gear := FALSE;
   Chain7Long.Drive.ACT.CMD.Enable := FALSE;
   Chain7Long.Drive.ACT.CMD.Pos_Mode := FALSE;
   Chain7Long.Drive.ACT.CMD.MergeDisabled := FALSE;
   Chain7Long.Drive.ACT.CMD.SCurve := FALSE;
   Chain7Long.Drive.ACT.CMD.Cam_Mode := TRUE;
   Chain7Long.Drive.ACT.CMD.Cam_Request := FALSE;
   Chain7Long.Drive.ACT.CMD.Cam_PhaseStop := FALSE;
   Chain7Long.Drive.ACT.CMD.Gear_Mode := FALSE;
   Chain7Long.Drive.ACT.CMD.Repos_Req := FALSE;
   Chain7Long.Drive.ACT.CMD.Jog_Pos := FALSE;
   Chain7Long.Drive.ACT.CMD.Jog_Neg := FALSE;
   Chain7Long.Drive.ACT.CMD.Stop := FALSE;
   Chain7Long.Drive.ACT.CMD.Calibration_Req := FALSE;
   Chain7Long.Drive.ACT.CMD.Reset := FALSE;
   Chain7Long.Drive.ACT.CMD.RegInput1 := FALSE;
   Chain7Long.Drive.ACT.CMD.Brake_Release := FALSE;
